// TwinCAT 3 PLC project DMMS_PLC
// ProgramVersion: 3.1.4026.19
// libraries:
//   Tc2_Standard, * (Beckhoff Automation GmbH)
//   Tc2_System, * (Beckhoff Automation GmbH)
//   Tc3_Mc3PlanarMotion, * (Beckhoff Automation GmbH)
//   Tc3_Physics, * (Beckhoff Automation GmbH)
//   Tc3_XPlanarStandard, * (Beckhoff Automation GmbH)
//   Tc3_XPlanarUtility, * (Beckhoff Automation GmbH)
// project tree:
//   DUTs/Communiction/GlobalStatus/ ST_ComIn_GlobalStatus.TcDUT (not stored), ST_ComOut_GlobalStatus.TcDUT (not stored), ST_Com_GlobalStatus.TcDUT (not stored)
//   DUTs/Communiction/Movers/ ST_ComIn_ExportMover.TcDUT, ST_ComOut_ExportMover.TcDUT, ST_PartTrackingData.TcDUT, ST_Com_ExportMover.TcDUT
//   DUTs/Communiction/Station/ ST_ComIn_ExportStation.TcDUT, ST_ComOut_ExportStation.TcDUT, ST_EStationName.TcDUT, ST_ManMov_Station.TcDUT, ST_Com_ExportStation.TcDUT
//   GVLs/ Communication.TcGVL, Debug.TcGVL (not stored), GVL.TcGVL
//   Mover/DUTs/ MoverPositionUnion.TcDUT (not stored), ST_ControlData.TcDUT, ST_EMoverLoadType.TcDUT, ST_ManMov_FreeMove.TcDUT (not stored), ST_ManMov_MoveTrack.TcDUT, ST_ManualMovements.TcDUT (not stored), ST_MoverConfiguration.TcDUT (not stored), ST_ProcessResult.TcDUT (not stored), ST_ProcessTask.TcDUT, ST_ProductData.TcDUT, ST_WellplateParametrization.TcDUT
//   Mover/ FB_ApplicationMover.TcPOU, I_MoverApplication.TcIO
//   / PlcTask.TcTTO (not stored)
//   POUs/ FB_MotionSystem.TcPOU, MAIN.TcPOU
//   Stations/Base/ FB_StationBase.TcPOU, I_Station.TcIO
//   Stations/DUTs/ E_ProcessMode.TcDUT (not stored), ST_EStationProcessState.TcDUT, ST_EStationHandshake.TcDUT (not stored), ST_StationPosition.TcDUT, ST_StationReturn.TcDUT (not stored), ST_VisStationData.TcDUT
//   Stations/ FB_PuncherStation.TcPOU, FB_PuncherSeparateStation.TcPOU (not stored), FB_PuncherBufferStation.TcPOU (not stored)
//   Stations/Helper/ FB_HistoryInfo.TcPOU (not stored)
//   Tracks/Base/ FB_BaseTrack.TcPOU (not stored), I_Track.TcIO (not stored)
//   Tracks/ FB_CloseLoopTrack.TcPOU, FB_UserInteractionTrack.TcPOU (not stored), FB_PipettePreBufferTrack.TcPOU (not stored), FB_PipetteTrack.TcPOU, FB_PipettePostBufferTrack.TcPOU (not stored), FB_PipetteBufferConTrack.TcPOU (not stored), FB_PuncherWellplateTrack.TcPOU (not stored), FB_PuncherBufferTrack.TcPOU, FB_StradeFirstSegTrack.TcPOU (not stored), FB_StradeSecondSegTrack.TcPOU (not stored), FB_PuncherSeperateTrack.TcPOU (not stored)
// real-time tasks:
//   TASK Job Task: cycle default, priority 2
//   TASK MC-Task (MET): cycle T#2ms, priority 3, ADS port 351
//   TASK MC-Task (MPT): cycle T#10ms, priority 4, ADS port 352
//   TASK PlcTask: cycle T#10ms, priority 20, ADS port 353
//   TASK XPlanar Task_0: cycle T#250us, priority 1, ADS port 350
//   TASK XPlanar Task_10: cycle T#250us, priority 5, ADS port 354
// I/O:
//   DEVICE Device 2 (EtherCAT), AmsNetId 192.168.2.44.3.1
//     Term 1 (APS4322-7000) [APS4322-7000 Drive]
//       Term 2 (APS4322-5000) [APS4322-5000 Feedback]
//     Term 3 (APS4322-7000) [APS4322-7000 Drive]
//       Term 4 (APS4322-5000) [APS4322-5000 Feedback]
//     Term 5 (APS4322-7000) [APS4322-7000 Drive]
//       Term 6 (APS4322-5000) [APS4322-5000 Feedback]
//     Term 7 (APS4322-7000) [APS4322-7000 Drive]
//       Term 8 (APS4322-5000) [APS4322-5000 Feedback]
//     Term 9 (APS4322-7000) [APS4322-7000 Drive]
//       Term 10 (APS4322-5000) [APS4322-5000 Feedback]
// variable links:
//   Device 2 (EtherCAT) <-> TcCOM Objects/XPlanar/Part1/APS4322_P1_1
//     Term 1 (APS4322-7000)/APS Comm Inputs/CommStatusWord <-> Data Pointer/MoverCommStatusWord
//     Term 1 (APS4322-7000)/APS Comm Inputs/Data {1..4} <-> Data Pointer/MoverCommDataIn[{0..3}]  (4 links)
//     Term 1 (APS4322-7000)/APS Comm Outputs/CommControlWord <-> Data Pointer/MoverCommControlWord
//     Term 1 (APS4322-7000)/APS Comm Outputs/Data 1 <-> Data Pointer/MoverCommDataOut
//     Term 1 (APS4322-7000)/APS Diagdata/DC Link Voltage <-> Data Pointer/DcLinkVoltage
//     Term 1 (APS4322-7000)/APS Diagdata/Power supply current <-> Data Pointer/PowerSupplyCurrent
//     Term 1 (APS4322-7000)/APS Inputs/StatusWord <-> Data Pointer/PowerUnitStatusWord
//     Term 1 (APS4322-7000)/APS Outputs/ControlWord <-> Data Pointer/PowerUnitControlWord
//     Term 1 (APS4322-7000)/APS Outputs/Current D 0X0 <-> Data Pointer/DCurrentSetPoints[0]
//     Term 1 (APS4322-7000)/APS Outputs/Current D 0X1 <-> Data Pointer/DCurrentSetPoints[1]
//     Term 1 (APS4322-7000)/APS Outputs/Current D 0X2 <-> Data Pointer/DCurrentSetPoints[2]
//     Term 1 (APS4322-7000)/APS Outputs/Current D 1X0 <-> Data Pointer/DCurrentSetPoints[6]
//     Term 1 (APS4322-7000)/APS Outputs/Current D 1X1 <-> Data Pointer/DCurrentSetPoints[7]
//     Term 1 (APS4322-7000)/APS Outputs/Current D 1X2 <-> Data Pointer/DCurrentSetPoints[8]
//     Term 1 (APS4322-7000)/APS Outputs/Current D 2X0 <-> Data Pointer/DCurrentSetPoints[12]
//     Term 1 (APS4322-7000)/APS Outputs/Current D 2X1 <-> Data Pointer/DCurrentSetPoints[13]
//     Term 1 (APS4322-7000)/APS Outputs/Current D 2X2 <-> Data Pointer/DCurrentSetPoints[14]
//     Term 1 (APS4322-7000)/APS Outputs/Current D 3X0 <-> Data Pointer/DCurrentSetPoints[18]
//     Term 1 (APS4322-7000)/APS Outputs/Current D 3X1 <-> Data Pointer/DCurrentSetPoints[19]
//     Term 1 (APS4322-7000)/APS Outputs/Current D 3X2 <-> Data Pointer/DCurrentSetPoints[20]
//     Term 1 (APS4322-7000)/APS Outputs/Current D 0Y0 <-> Data Pointer/DCurrentSetPoints[3]
//     Term 1 (APS4322-7000)/APS Outputs/Current D 0Y1 <-> Data Pointer/DCurrentSetPoints[4]
//     Term 1 (APS4322-7000)/APS Outputs/Current D 0Y2 <-> Data Pointer/DCurrentSetPoints[5]
//     Term 1 (APS4322-7000)/APS Outputs/Current D 1Y0 <-> Data Pointer/DCurrentSetPoints[9]
//     Term 1 (APS4322-7000)/APS Outputs/Current D 1Y1 <-> Data Pointer/DCurrentSetPoints[10]
//     Term 1 (APS4322-7000)/APS Outputs/Current D 1Y2 <-> Data Pointer/DCurrentSetPoints[11]
//     Term 1 (APS4322-7000)/APS Outputs/Current D 2Y0 <-> Data Pointer/DCurrentSetPoints[15]
//     Term 1 (APS4322-7000)/APS Outputs/Current D 2Y1 <-> Data Pointer/DCurrentSetPoints[16]
//     Term 1 (APS4322-7000)/APS Outputs/Current D 2Y2 <-> Data Pointer/DCurrentSetPoints[17]
//     Term 1 (APS4322-7000)/APS Outputs/Current D 3Y0 <-> Data Pointer/DCurrentSetPoints[21]
//     Term 1 (APS4322-7000)/APS Outputs/Current D 3Y1 <-> Data Pointer/DCurrentSetPoints[22]
//     Term 1 (APS4322-7000)/APS Outputs/Current D 3Y2 <-> Data Pointer/DCurrentSetPoints[23]
//     Term 1 (APS4322-7000)/APS Outputs/Current Q 0X0 <-> Data Pointer/QCurrentSetPoints[0]
//     Term 1 (APS4322-7000)/APS Outputs/Current Q 0X1 <-> Data Pointer/QCurrentSetPoints[1]
//     Term 1 (APS4322-7000)/APS Outputs/Current Q 0X2 <-> Data Pointer/QCurrentSetPoints[2]
//     Term 1 (APS4322-7000)/APS Outputs/Current Q 1X0 <-> Data Pointer/QCurrentSetPoints[6]
//     Term 1 (APS4322-7000)/APS Outputs/Current Q 1X1 <-> Data Pointer/QCurrentSetPoints[7]
//     Term 1 (APS4322-7000)/APS Outputs/Current Q 1X2 <-> Data Pointer/QCurrentSetPoints[8]
//     Term 1 (APS4322-7000)/APS Outputs/Current Q 2X0 <-> Data Pointer/QCurrentSetPoints[12]
//     Term 1 (APS4322-7000)/APS Outputs/Current Q 2X1 <-> Data Pointer/QCurrentSetPoints[13]
//     Term 1 (APS4322-7000)/APS Outputs/Current Q 2X2 <-> Data Pointer/QCurrentSetPoints[14]
//     Term 1 (APS4322-7000)/APS Outputs/Current Q 3X0 <-> Data Pointer/QCurrentSetPoints[18]
//     Term 1 (APS4322-7000)/APS Outputs/Current Q 3X1 <-> Data Pointer/QCurrentSetPoints[19]
//     Term 1 (APS4322-7000)/APS Outputs/Current Q 3X2 <-> Data Pointer/QCurrentSetPoints[20]
//     Term 1 (APS4322-7000)/APS Outputs/Current Q 0Y0 <-> Data Pointer/QCurrentSetPoints[3]
//     Term 1 (APS4322-7000)/APS Outputs/Current Q 0Y1 <-> Data Pointer/QCurrentSetPoints[4]
//     Term 1 (APS4322-7000)/APS Outputs/Current Q 0Y2 <-> Data Pointer/QCurrentSetPoints[5]
//     Term 1 (APS4322-7000)/APS Outputs/Current Q 1Y0 <-> Data Pointer/QCurrentSetPoints[9]
//     Term 1 (APS4322-7000)/APS Outputs/Current Q 1Y1 <-> Data Pointer/QCurrentSetPoints[10]
//     Term 1 (APS4322-7000)/APS Outputs/Current Q 1Y2 <-> Data Pointer/QCurrentSetPoints[11]
//     Term 1 (APS4322-7000)/APS Outputs/Current Q 2Y0 <-> Data Pointer/QCurrentSetPoints[15]
//     Term 1 (APS4322-7000)/APS Outputs/Current Q 2Y1 <-> Data Pointer/QCurrentSetPoints[16]
//     Term 1 (APS4322-7000)/APS Outputs/Current Q 2Y2 <-> Data Pointer/QCurrentSetPoints[17]
//     Term 1 (APS4322-7000)/APS Outputs/Current Q 3Y0 <-> Data Pointer/QCurrentSetPoints[21]
//     Term 1 (APS4322-7000)/APS Outputs/Current Q 3Y1 <-> Data Pointer/QCurrentSetPoints[22]
//     Term 1 (APS4322-7000)/APS Outputs/Current Q 3Y2 <-> Data Pointer/QCurrentSetPoints[23]
//     Term 1 (APS4322-7000)/APS Outputs/PhiE 0X0 <-> Data Pointer/PhiSetPoints[0]
//     Term 1 (APS4322-7000)/APS Outputs/PhiE 0X1 <-> Data Pointer/PhiSetPoints[1]
//     Term 1 (APS4322-7000)/APS Outputs/PhiE 0X2 <-> Data Pointer/PhiSetPoints[2]
//     Term 1 (APS4322-7000)/APS Outputs/PhiE 1X0 <-> Data Pointer/PhiSetPoints[6]
//     Term 1 (APS4322-7000)/APS Outputs/PhiE 1X1 <-> Data Pointer/PhiSetPoints[7]
//     Term 1 (APS4322-7000)/APS Outputs/PhiE 1X2 <-> Data Pointer/PhiSetPoints[8]
//     Term 1 (APS4322-7000)/APS Outputs/PhiE 2X0 <-> Data Pointer/PhiSetPoints[12]
//     Term 1 (APS4322-7000)/APS Outputs/PhiE 2X1 <-> Data Pointer/PhiSetPoints[13]
//     Term 1 (APS4322-7000)/APS Outputs/PhiE 2X2 <-> Data Pointer/PhiSetPoints[14]
//     Term 1 (APS4322-7000)/APS Outputs/PhiE 3X0 <-> Data Pointer/PhiSetPoints[18]
//     Term 1 (APS4322-7000)/APS Outputs/PhiE 3X1 <-> Data Pointer/PhiSetPoints[19]
//     Term 1 (APS4322-7000)/APS Outputs/PhiE 3X2 <-> Data Pointer/PhiSetPoints[20]
//     Term 1 (APS4322-7000)/APS Outputs/PhiE 0Y0 <-> Data Pointer/PhiSetPoints[3]
//     Term 1 (APS4322-7000)/APS Outputs/PhiE 0Y1 <-> Data Pointer/PhiSetPoints[4]
//     Term 1 (APS4322-7000)/APS Outputs/PhiE 0Y2 <-> Data Pointer/PhiSetPoints[5]
//     Term 1 (APS4322-7000)/APS Outputs/PhiE 1Y0 <-> Data Pointer/PhiSetPoints[9]
//     Term 1 (APS4322-7000)/APS Outputs/PhiE 1Y1 <-> Data Pointer/PhiSetPoints[10]
//     Term 1 (APS4322-7000)/APS Outputs/PhiE 1Y2 <-> Data Pointer/PhiSetPoints[11]
//     Term 1 (APS4322-7000)/APS Outputs/PhiE 2Y0 <-> Data Pointer/PhiSetPoints[15]
//     Term 1 (APS4322-7000)/APS Outputs/PhiE 2Y1 <-> Data Pointer/PhiSetPoints[16]
//     Term 1 (APS4322-7000)/APS Outputs/PhiE 2Y2 <-> Data Pointer/PhiSetPoints[17]
//     Term 1 (APS4322-7000)/APS Outputs/PhiE 3Y0 <-> Data Pointer/PhiSetPoints[21]
//     Term 1 (APS4322-7000)/APS Outputs/PhiE 3Y1 <-> Data Pointer/PhiSetPoints[22]
//     Term 1 (APS4322-7000)/APS Outputs/PhiE 3Y2 <-> Data Pointer/PhiSetPoints[23]
//     Term 1 (APS4322-7000)/Term 2 (APS4322-5000)/FB Inputs/A{0..8 step 2} X-Field <-> Data Pointer/HallSensorFieldsXYZ[{0..12 step 3}]  (5 links)
//     Term 1 (APS4322-7000)/Term 2 (APS4322-5000)/FB Inputs/A{0..8 step 2} Y-Field <-> Data Pointer/HallSensorFieldsXYZ[{1..13 step 3}]  (5 links)
//     Term 1 (APS4322-7000)/Term 2 (APS4322-5000)/FB Inputs/A{0..8 step 2} Z-Field <-> Data Pointer/HallSensorFieldsXYZ[{2..14 step 3}]  (5 links)
//     Term 1 (APS4322-7000)/Term 2 (APS4322-5000)/FB Inputs/B{1..9 step 2} X-Field <-> Data Pointer/HallSensorFieldsXYZ[{15..27 step 3}]  (5 links)
//     Term 1 (APS4322-7000)/Term 2 (APS4322-5000)/FB Inputs/B{1..9 step 2} Y-Field <-> Data Pointer/HallSensorFieldsXYZ[{16..28 step 3}]  (5 links)
//     Term 1 (APS4322-7000)/Term 2 (APS4322-5000)/FB Inputs/B{1..9 step 2} Z-Field <-> Data Pointer/HallSensorFieldsXYZ[{17..29 step 3}]  (5 links)
//     Term 1 (APS4322-7000)/Term 2 (APS4322-5000)/FB Inputs/C{0..8 step 2} X-Field <-> Data Pointer/HallSensorFieldsXYZ[{30..42 step 3}]  (5 links)
//     Term 1 (APS4322-7000)/Term 2 (APS4322-5000)/FB Inputs/C{0..8 step 2} Y-Field <-> Data Pointer/HallSensorFieldsXYZ[{31..43 step 3}]  (5 links)
//     Term 1 (APS4322-7000)/Term 2 (APS4322-5000)/FB Inputs/C{0..8 step 2} Z-Field <-> Data Pointer/HallSensorFieldsXYZ[{32..44 step 3}]  (5 links)
//     Term 1 (APS4322-7000)/Term 2 (APS4322-5000)/FB Inputs/D{1..9 step 2} X-Field <-> Data Pointer/HallSensorFieldsXYZ[{45..57 step 3}]  (5 links)
//     Term 1 (APS4322-7000)/Term 2 (APS4322-5000)/FB Inputs/D{1..9 step 2} Y-Field <-> Data Pointer/HallSensorFieldsXYZ[{46..58 step 3}]  (5 links)
//     Term 1 (APS4322-7000)/Term 2 (APS4322-5000)/FB Inputs/D{1..9 step 2} Z-Field <-> Data Pointer/HallSensorFieldsXYZ[{47..59 step 3}]  (5 links)
//     Term 1 (APS4322-7000)/Term 2 (APS4322-5000)/FB Inputs/E{0..8 step 2} X-Field <-> Data Pointer/HallSensorFieldsXYZ[{60..72 step 3}]  (5 links)
//     Term 1 (APS4322-7000)/Term 2 (APS4322-5000)/FB Inputs/E{0..8 step 2} Y-Field <-> Data Pointer/HallSensorFieldsXYZ[{61..73 step 3}]  (5 links)
//     Term 1 (APS4322-7000)/Term 2 (APS4322-5000)/FB Inputs/E{0..8 step 2} Z-Field <-> Data Pointer/HallSensorFieldsXYZ[{62..74 step 3}]  (5 links)
//     Term 1 (APS4322-7000)/Term 2 (APS4322-5000)/FB Inputs/F{1..9 step 2} X-Field <-> Data Pointer/HallSensorFieldsXYZ[{75..87 step 3}]  (5 links)
//     Term 1 (APS4322-7000)/Term 2 (APS4322-5000)/FB Inputs/F{1..9 step 2} Y-Field <-> Data Pointer/HallSensorFieldsXYZ[{76..88 step 3}]  (5 links)
//     Term 1 (APS4322-7000)/Term 2 (APS4322-5000)/FB Inputs/F{1..9 step 2} Z-Field <-> Data Pointer/HallSensorFieldsXYZ[{77..89 step 3}]  (5 links)
//     Term 1 (APS4322-7000)/Term 2 (APS4322-5000)/FB Inputs/G{0..8 step 2} X-Field <-> Data Pointer/HallSensorFieldsXYZ[{90..102 step 3}]  (5 links)
//     Term 1 (APS4322-7000)/Term 2 (APS4322-5000)/FB Inputs/G{0..8 step 2} Y-Field <-> Data Pointer/HallSensorFieldsXYZ[{91..103 step 3}]  (5 links)
//     Term 1 (APS4322-7000)/Term 2 (APS4322-5000)/FB Inputs/G{0..8 step 2} Z-Field <-> Data Pointer/HallSensorFieldsXYZ[{92..104 step 3}]  (5 links)
//     Term 1 (APS4322-7000)/Term 2 (APS4322-5000)/FB Inputs/H{1..9 step 2} X-Field <-> Data Pointer/HallSensorFieldsXYZ[{105..117 step 3}]  (5 links)
//     Term 1 (APS4322-7000)/Term 2 (APS4322-5000)/FB Inputs/H{1..9 step 2} Y-Field <-> Data Pointer/HallSensorFieldsXYZ[{106..118 step 3}]  (5 links)
//     Term 1 (APS4322-7000)/Term 2 (APS4322-5000)/FB Inputs/H{1..9 step 2} Z-Field <-> Data Pointer/HallSensorFieldsXYZ[{107..119 step 3}]  (5 links)
//     Term 1 (APS4322-7000)/Term 2 (APS4322-5000)/FB Inputs/I{0..8 step 2} X-Field <-> Data Pointer/HallSensorFieldsXYZ[{120..132 step 3}]  (5 links)
//     Term 1 (APS4322-7000)/Term 2 (APS4322-5000)/FB Inputs/I{0..8 step 2} Y-Field <-> Data Pointer/HallSensorFieldsXYZ[{121..133 step 3}]  (5 links)
//     Term 1 (APS4322-7000)/Term 2 (APS4322-5000)/FB Inputs/I{0..8 step 2} Z-Field <-> Data Pointer/HallSensorFieldsXYZ[{122..134 step 3}]  (5 links)
//     Term 1 (APS4322-7000)/Term 2 (APS4322-5000)/FB Inputs/J{1..9 step 2} X-Field <-> Data Pointer/HallSensorFieldsXYZ[{135..147 step 3}]  (5 links)
//     Term 1 (APS4322-7000)/Term 2 (APS4322-5000)/FB Inputs/J{1..9 step 2} Y-Field <-> Data Pointer/HallSensorFieldsXYZ[{136..148 step 3}]  (5 links)
//     Term 1 (APS4322-7000)/Term 2 (APS4322-5000)/FB Inputs/J{1..9 step 2} Z-Field <-> Data Pointer/HallSensorFieldsXYZ[{137..149 step 3}]  (5 links)
//     Term 1 (APS4322-7000)/Term 2 (APS4322-5000)/FB Inputs/Status <-> Data Pointer/FeedbackStatus
//   Device 2 (EtherCAT) <-> TcCOM Objects/XPlanar/Part1/APS4322_P1_2
//     Term 3 (APS4322-7000)/APS Comm Inputs/CommStatusWord <-> Data Pointer/MoverCommStatusWord
//     Term 3 (APS4322-7000)/APS Comm Inputs/Data {1..4} <-> Data Pointer/MoverCommDataIn[{0..3}]  (4 links)
//     Term 3 (APS4322-7000)/APS Comm Outputs/CommControlWord <-> Data Pointer/MoverCommControlWord
//     Term 3 (APS4322-7000)/APS Comm Outputs/Data 1 <-> Data Pointer/MoverCommDataOut
//     Term 3 (APS4322-7000)/APS Diagdata/DC Link Voltage <-> Data Pointer/DcLinkVoltage
//     Term 3 (APS4322-7000)/APS Diagdata/Power supply current <-> Data Pointer/PowerSupplyCurrent
//     Term 3 (APS4322-7000)/APS Inputs/StatusWord <-> Data Pointer/PowerUnitStatusWord
//     Term 3 (APS4322-7000)/APS Outputs/ControlWord <-> Data Pointer/PowerUnitControlWord
//     Term 3 (APS4322-7000)/APS Outputs/Current D 0X0 <-> Data Pointer/DCurrentSetPoints[0]
//     Term 3 (APS4322-7000)/APS Outputs/Current D 0X1 <-> Data Pointer/DCurrentSetPoints[1]
//     Term 3 (APS4322-7000)/APS Outputs/Current D 0X2 <-> Data Pointer/DCurrentSetPoints[2]
//     Term 3 (APS4322-7000)/APS Outputs/Current D 1X0 <-> Data Pointer/DCurrentSetPoints[6]
//     Term 3 (APS4322-7000)/APS Outputs/Current D 1X1 <-> Data Pointer/DCurrentSetPoints[7]
//     Term 3 (APS4322-7000)/APS Outputs/Current D 1X2 <-> Data Pointer/DCurrentSetPoints[8]
//     Term 3 (APS4322-7000)/APS Outputs/Current D 2X0 <-> Data Pointer/DCurrentSetPoints[12]
//     Term 3 (APS4322-7000)/APS Outputs/Current D 2X1 <-> Data Pointer/DCurrentSetPoints[13]
//     Term 3 (APS4322-7000)/APS Outputs/Current D 2X2 <-> Data Pointer/DCurrentSetPoints[14]
//     Term 3 (APS4322-7000)/APS Outputs/Current D 3X0 <-> Data Pointer/DCurrentSetPoints[18]
//     Term 3 (APS4322-7000)/APS Outputs/Current D 3X1 <-> Data Pointer/DCurrentSetPoints[19]
//     Term 3 (APS4322-7000)/APS Outputs/Current D 3X2 <-> Data Pointer/DCurrentSetPoints[20]
//     Term 3 (APS4322-7000)/APS Outputs/Current D 0Y0 <-> Data Pointer/DCurrentSetPoints[3]
//     Term 3 (APS4322-7000)/APS Outputs/Current D 0Y1 <-> Data Pointer/DCurrentSetPoints[4]
//     Term 3 (APS4322-7000)/APS Outputs/Current D 0Y2 <-> Data Pointer/DCurrentSetPoints[5]
//     Term 3 (APS4322-7000)/APS Outputs/Current D 1Y0 <-> Data Pointer/DCurrentSetPoints[9]
//     Term 3 (APS4322-7000)/APS Outputs/Current D 1Y1 <-> Data Pointer/DCurrentSetPoints[10]
//     Term 3 (APS4322-7000)/APS Outputs/Current D 1Y2 <-> Data Pointer/DCurrentSetPoints[11]
//     Term 3 (APS4322-7000)/APS Outputs/Current D 2Y0 <-> Data Pointer/DCurrentSetPoints[15]
//     Term 3 (APS4322-7000)/APS Outputs/Current D 2Y1 <-> Data Pointer/DCurrentSetPoints[16]
//     Term 3 (APS4322-7000)/APS Outputs/Current D 2Y2 <-> Data Pointer/DCurrentSetPoints[17]
//     Term 3 (APS4322-7000)/APS Outputs/Current D 3Y0 <-> Data Pointer/DCurrentSetPoints[21]
//     Term 3 (APS4322-7000)/APS Outputs/Current D 3Y1 <-> Data Pointer/DCurrentSetPoints[22]
//     Term 3 (APS4322-7000)/APS Outputs/Current D 3Y2 <-> Data Pointer/DCurrentSetPoints[23]
//     Term 3 (APS4322-7000)/APS Outputs/Current Q 0X0 <-> Data Pointer/QCurrentSetPoints[0]
//     Term 3 (APS4322-7000)/APS Outputs/Current Q 0X1 <-> Data Pointer/QCurrentSetPoints[1]
//     Term 3 (APS4322-7000)/APS Outputs/Current Q 0X2 <-> Data Pointer/QCurrentSetPoints[2]
//     Term 3 (APS4322-7000)/APS Outputs/Current Q 1X0 <-> Data Pointer/QCurrentSetPoints[6]
//     Term 3 (APS4322-7000)/APS Outputs/Current Q 1X1 <-> Data Pointer/QCurrentSetPoints[7]
//     Term 3 (APS4322-7000)/APS Outputs/Current Q 1X2 <-> Data Pointer/QCurrentSetPoints[8]
//     Term 3 (APS4322-7000)/APS Outputs/Current Q 2X0 <-> Data Pointer/QCurrentSetPoints[12]
//     Term 3 (APS4322-7000)/APS Outputs/Current Q 2X1 <-> Data Pointer/QCurrentSetPoints[13]
//     Term 3 (APS4322-7000)/APS Outputs/Current Q 2X2 <-> Data Pointer/QCurrentSetPoints[14]
//     Term 3 (APS4322-7000)/APS Outputs/Current Q 3X0 <-> Data Pointer/QCurrentSetPoints[18]
//     Term 3 (APS4322-7000)/APS Outputs/Current Q 3X1 <-> Data Pointer/QCurrentSetPoints[19]
//     Term 3 (APS4322-7000)/APS Outputs/Current Q 3X2 <-> Data Pointer/QCurrentSetPoints[20]
//     Term 3 (APS4322-7000)/APS Outputs/Current Q 0Y0 <-> Data Pointer/QCurrentSetPoints[3]
//     Term 3 (APS4322-7000)/APS Outputs/Current Q 0Y1 <-> Data Pointer/QCurrentSetPoints[4]
//     Term 3 (APS4322-7000)/APS Outputs/Current Q 0Y2 <-> Data Pointer/QCurrentSetPoints[5]
//     Term 3 (APS4322-7000)/APS Outputs/Current Q 1Y0 <-> Data Pointer/QCurrentSetPoints[9]
//     Term 3 (APS4322-7000)/APS Outputs/Current Q 1Y1 <-> Data Pointer/QCurrentSetPoints[10]
//     Term 3 (APS4322-7000)/APS Outputs/Current Q 1Y2 <-> Data Pointer/QCurrentSetPoints[11]
//     Term 3 (APS4322-7000)/APS Outputs/Current Q 2Y0 <-> Data Pointer/QCurrentSetPoints[15]
//     Term 3 (APS4322-7000)/APS Outputs/Current Q 2Y1 <-> Data Pointer/QCurrentSetPoints[16]
//     Term 3 (APS4322-7000)/APS Outputs/Current Q 2Y2 <-> Data Pointer/QCurrentSetPoints[17]
//     Term 3 (APS4322-7000)/APS Outputs/Current Q 3Y0 <-> Data Pointer/QCurrentSetPoints[21]
//     Term 3 (APS4322-7000)/APS Outputs/Current Q 3Y1 <-> Data Pointer/QCurrentSetPoints[22]
//     Term 3 (APS4322-7000)/APS Outputs/Current Q 3Y2 <-> Data Pointer/QCurrentSetPoints[23]
//     Term 3 (APS4322-7000)/APS Outputs/PhiE 0X0 <-> Data Pointer/PhiSetPoints[0]
//     Term 3 (APS4322-7000)/APS Outputs/PhiE 0X1 <-> Data Pointer/PhiSetPoints[1]
//     Term 3 (APS4322-7000)/APS Outputs/PhiE 0X2 <-> Data Pointer/PhiSetPoints[2]
//     Term 3 (APS4322-7000)/APS Outputs/PhiE 1X0 <-> Data Pointer/PhiSetPoints[6]
//     Term 3 (APS4322-7000)/APS Outputs/PhiE 1X1 <-> Data Pointer/PhiSetPoints[7]
//     Term 3 (APS4322-7000)/APS Outputs/PhiE 1X2 <-> Data Pointer/PhiSetPoints[8]
//     Term 3 (APS4322-7000)/APS Outputs/PhiE 2X0 <-> Data Pointer/PhiSetPoints[12]
//     Term 3 (APS4322-7000)/APS Outputs/PhiE 2X1 <-> Data Pointer/PhiSetPoints[13]
//     Term 3 (APS4322-7000)/APS Outputs/PhiE 2X2 <-> Data Pointer/PhiSetPoints[14]
//     Term 3 (APS4322-7000)/APS Outputs/PhiE 3X0 <-> Data Pointer/PhiSetPoints[18]
//     Term 3 (APS4322-7000)/APS Outputs/PhiE 3X1 <-> Data Pointer/PhiSetPoints[19]
//     Term 3 (APS4322-7000)/APS Outputs/PhiE 3X2 <-> Data Pointer/PhiSetPoints[20]
//     Term 3 (APS4322-7000)/APS Outputs/PhiE 0Y0 <-> Data Pointer/PhiSetPoints[3]
//     Term 3 (APS4322-7000)/APS Outputs/PhiE 0Y1 <-> Data Pointer/PhiSetPoints[4]
//     Term 3 (APS4322-7000)/APS Outputs/PhiE 0Y2 <-> Data Pointer/PhiSetPoints[5]
//     Term 3 (APS4322-7000)/APS Outputs/PhiE 1Y0 <-> Data Pointer/PhiSetPoints[9]
//     Term 3 (APS4322-7000)/APS Outputs/PhiE 1Y1 <-> Data Pointer/PhiSetPoints[10]
//     Term 3 (APS4322-7000)/APS Outputs/PhiE 1Y2 <-> Data Pointer/PhiSetPoints[11]
//     Term 3 (APS4322-7000)/APS Outputs/PhiE 2Y0 <-> Data Pointer/PhiSetPoints[15]
//     Term 3 (APS4322-7000)/APS Outputs/PhiE 2Y1 <-> Data Pointer/PhiSetPoints[16]
//     Term 3 (APS4322-7000)/APS Outputs/PhiE 2Y2 <-> Data Pointer/PhiSetPoints[17]
//     Term 3 (APS4322-7000)/APS Outputs/PhiE 3Y0 <-> Data Pointer/PhiSetPoints[21]
//     Term 3 (APS4322-7000)/APS Outputs/PhiE 3Y1 <-> Data Pointer/PhiSetPoints[22]
//     Term 3 (APS4322-7000)/APS Outputs/PhiE 3Y2 <-> Data Pointer/PhiSetPoints[23]
//     Term 3 (APS4322-7000)/Term 4 (APS4322-5000)/FB Inputs/A{0..8 step 2} X-Field <-> Data Pointer/HallSensorFieldsXYZ[{0..12 step 3}]  (5 links)
//     Term 3 (APS4322-7000)/Term 4 (APS4322-5000)/FB Inputs/A{0..8 step 2} Y-Field <-> Data Pointer/HallSensorFieldsXYZ[{1..13 step 3}]  (5 links)
//     Term 3 (APS4322-7000)/Term 4 (APS4322-5000)/FB Inputs/A{0..8 step 2} Z-Field <-> Data Pointer/HallSensorFieldsXYZ[{2..14 step 3}]  (5 links)
//     Term 3 (APS4322-7000)/Term 4 (APS4322-5000)/FB Inputs/B{1..9 step 2} X-Field <-> Data Pointer/HallSensorFieldsXYZ[{15..27 step 3}]  (5 links)
//     Term 3 (APS4322-7000)/Term 4 (APS4322-5000)/FB Inputs/B{1..9 step 2} Y-Field <-> Data Pointer/HallSensorFieldsXYZ[{16..28 step 3}]  (5 links)
//     Term 3 (APS4322-7000)/Term 4 (APS4322-5000)/FB Inputs/B{1..9 step 2} Z-Field <-> Data Pointer/HallSensorFieldsXYZ[{17..29 step 3}]  (5 links)
//     Term 3 (APS4322-7000)/Term 4 (APS4322-5000)/FB Inputs/C{0..8 step 2} X-Field <-> Data Pointer/HallSensorFieldsXYZ[{30..42 step 3}]  (5 links)
//     Term 3 (APS4322-7000)/Term 4 (APS4322-5000)/FB Inputs/C{0..8 step 2} Y-Field <-> Data Pointer/HallSensorFieldsXYZ[{31..43 step 3}]  (5 links)
//     Term 3 (APS4322-7000)/Term 4 (APS4322-5000)/FB Inputs/C{0..8 step 2} Z-Field <-> Data Pointer/HallSensorFieldsXYZ[{32..44 step 3}]  (5 links)
//     Term 3 (APS4322-7000)/Term 4 (APS4322-5000)/FB Inputs/D{1..9 step 2} X-Field <-> Data Pointer/HallSensorFieldsXYZ[{45..57 step 3}]  (5 links)
//     Term 3 (APS4322-7000)/Term 4 (APS4322-5000)/FB Inputs/D{1..9 step 2} Y-Field <-> Data Pointer/HallSensorFieldsXYZ[{46..58 step 3}]  (5 links)
//     Term 3 (APS4322-7000)/Term 4 (APS4322-5000)/FB Inputs/D{1..9 step 2} Z-Field <-> Data Pointer/HallSensorFieldsXYZ[{47..59 step 3}]  (5 links)
//     Term 3 (APS4322-7000)/Term 4 (APS4322-5000)/FB Inputs/E{0..8 step 2} X-Field <-> Data Pointer/HallSensorFieldsXYZ[{60..72 step 3}]  (5 links)
//     Term 3 (APS4322-7000)/Term 4 (APS4322-5000)/FB Inputs/E{0..8 step 2} Y-Field <-> Data Pointer/HallSensorFieldsXYZ[{61..73 step 3}]  (5 links)
//     Term 3 (APS4322-7000)/Term 4 (APS4322-5000)/FB Inputs/E{0..8 step 2} Z-Field <-> Data Pointer/HallSensorFieldsXYZ[{62..74 step 3}]  (5 links)
//     Term 3 (APS4322-7000)/Term 4 (APS4322-5000)/FB Inputs/F{1..9 step 2} X-Field <-> Data Pointer/HallSensorFieldsXYZ[{75..87 step 3}]  (5 links)
//     Term 3 (APS4322-7000)/Term 4 (APS4322-5000)/FB Inputs/F{1..9 step 2} Y-Field <-> Data Pointer/HallSensorFieldsXYZ[{76..88 step 3}]  (5 links)
//     Term 3 (APS4322-7000)/Term 4 (APS4322-5000)/FB Inputs/F{1..9 step 2} Z-Field <-> Data Pointer/HallSensorFieldsXYZ[{77..89 step 3}]  (5 links)
//     Term 3 (APS4322-7000)/Term 4 (APS4322-5000)/FB Inputs/G{0..8 step 2} X-Field <-> Data Pointer/HallSensorFieldsXYZ[{90..102 step 3}]  (5 links)
//     Term 3 (APS4322-7000)/Term 4 (APS4322-5000)/FB Inputs/G{0..8 step 2} Y-Field <-> Data Pointer/HallSensorFieldsXYZ[{91..103 step 3}]  (5 links)
//     Term 3 (APS4322-7000)/Term 4 (APS4322-5000)/FB Inputs/G{0..8 step 2} Z-Field <-> Data Pointer/HallSensorFieldsXYZ[{92..104 step 3}]  (5 links)
//     Term 3 (APS4322-7000)/Term 4 (APS4322-5000)/FB Inputs/H{1..9 step 2} X-Field <-> Data Pointer/HallSensorFieldsXYZ[{105..117 step 3}]  (5 links)
//     Term 3 (APS4322-7000)/Term 4 (APS4322-5000)/FB Inputs/H{1..9 step 2} Y-Field <-> Data Pointer/HallSensorFieldsXYZ[{106..118 step 3}]  (5 links)
//     Term 3 (APS4322-7000)/Term 4 (APS4322-5000)/FB Inputs/H{1..9 step 2} Z-Field <-> Data Pointer/HallSensorFieldsXYZ[{107..119 step 3}]  (5 links)
//     Term 3 (APS4322-7000)/Term 4 (APS4322-5000)/FB Inputs/I{0..8 step 2} X-Field <-> Data Pointer/HallSensorFieldsXYZ[{120..132 step 3}]  (5 links)
//     Term 3 (APS4322-7000)/Term 4 (APS4322-5000)/FB Inputs/I{0..8 step 2} Y-Field <-> Data Pointer/HallSensorFieldsXYZ[{121..133 step 3}]  (5 links)
//     Term 3 (APS4322-7000)/Term 4 (APS4322-5000)/FB Inputs/I{0..8 step 2} Z-Field <-> Data Pointer/HallSensorFieldsXYZ[{122..134 step 3}]  (5 links)
//     Term 3 (APS4322-7000)/Term 4 (APS4322-5000)/FB Inputs/J{1..9 step 2} X-Field <-> Data Pointer/HallSensorFieldsXYZ[{135..147 step 3}]  (5 links)
//     Term 3 (APS4322-7000)/Term 4 (APS4322-5000)/FB Inputs/J{1..9 step 2} Y-Field <-> Data Pointer/HallSensorFieldsXYZ[{136..148 step 3}]  (5 links)
//     Term 3 (APS4322-7000)/Term 4 (APS4322-5000)/FB Inputs/J{1..9 step 2} Z-Field <-> Data Pointer/HallSensorFieldsXYZ[{137..149 step 3}]  (5 links)
//     Term 3 (APS4322-7000)/Term 4 (APS4322-5000)/FB Inputs/Status <-> Data Pointer/FeedbackStatus
//   Device 2 (EtherCAT) <-> TcCOM Objects/XPlanar/Part1/APS4322_P1_3
//     Term 5 (APS4322-7000)/APS Comm Inputs/CommStatusWord <-> Data Pointer/MoverCommStatusWord
//     Term 5 (APS4322-7000)/APS Comm Inputs/Data {1..4} <-> Data Pointer/MoverCommDataIn[{0..3}]  (4 links)
//     Term 5 (APS4322-7000)/APS Comm Outputs/CommControlWord <-> Data Pointer/MoverCommControlWord
//     Term 5 (APS4322-7000)/APS Comm Outputs/Data 1 <-> Data Pointer/MoverCommDataOut
//     Term 5 (APS4322-7000)/APS Diagdata/DC Link Voltage <-> Data Pointer/DcLinkVoltage
//     Term 5 (APS4322-7000)/APS Diagdata/Power supply current <-> Data Pointer/PowerSupplyCurrent
//     Term 5 (APS4322-7000)/APS Inputs/StatusWord <-> Data Pointer/PowerUnitStatusWord
//     Term 5 (APS4322-7000)/APS Outputs/ControlWord <-> Data Pointer/PowerUnitControlWord
//     Term 5 (APS4322-7000)/APS Outputs/Current D 0X0 <-> Data Pointer/DCurrentSetPoints[0]
//     Term 5 (APS4322-7000)/APS Outputs/Current D 0X1 <-> Data Pointer/DCurrentSetPoints[1]
//     Term 5 (APS4322-7000)/APS Outputs/Current D 0X2 <-> Data Pointer/DCurrentSetPoints[2]
//     Term 5 (APS4322-7000)/APS Outputs/Current D 1X0 <-> Data Pointer/DCurrentSetPoints[6]
//     Term 5 (APS4322-7000)/APS Outputs/Current D 1X1 <-> Data Pointer/DCurrentSetPoints[7]
//     Term 5 (APS4322-7000)/APS Outputs/Current D 1X2 <-> Data Pointer/DCurrentSetPoints[8]
//     Term 5 (APS4322-7000)/APS Outputs/Current D 2X0 <-> Data Pointer/DCurrentSetPoints[12]
//     Term 5 (APS4322-7000)/APS Outputs/Current D 2X1 <-> Data Pointer/DCurrentSetPoints[13]
//     Term 5 (APS4322-7000)/APS Outputs/Current D 2X2 <-> Data Pointer/DCurrentSetPoints[14]
//     Term 5 (APS4322-7000)/APS Outputs/Current D 3X0 <-> Data Pointer/DCurrentSetPoints[18]
//     Term 5 (APS4322-7000)/APS Outputs/Current D 3X1 <-> Data Pointer/DCurrentSetPoints[19]
//     Term 5 (APS4322-7000)/APS Outputs/Current D 3X2 <-> Data Pointer/DCurrentSetPoints[20]
//     Term 5 (APS4322-7000)/APS Outputs/Current D 0Y0 <-> Data Pointer/DCurrentSetPoints[3]
//     Term 5 (APS4322-7000)/APS Outputs/Current D 0Y1 <-> Data Pointer/DCurrentSetPoints[4]
//     Term 5 (APS4322-7000)/APS Outputs/Current D 0Y2 <-> Data Pointer/DCurrentSetPoints[5]
//     Term 5 (APS4322-7000)/APS Outputs/Current D 1Y0 <-> Data Pointer/DCurrentSetPoints[9]
//     Term 5 (APS4322-7000)/APS Outputs/Current D 1Y1 <-> Data Pointer/DCurrentSetPoints[10]
//     Term 5 (APS4322-7000)/APS Outputs/Current D 1Y2 <-> Data Pointer/DCurrentSetPoints[11]
//     Term 5 (APS4322-7000)/APS Outputs/Current D 2Y0 <-> Data Pointer/DCurrentSetPoints[15]
//     Term 5 (APS4322-7000)/APS Outputs/Current D 2Y1 <-> Data Pointer/DCurrentSetPoints[16]
//     Term 5 (APS4322-7000)/APS Outputs/Current D 2Y2 <-> Data Pointer/DCurrentSetPoints[17]
//     Term 5 (APS4322-7000)/APS Outputs/Current D 3Y0 <-> Data Pointer/DCurrentSetPoints[21]
//     Term 5 (APS4322-7000)/APS Outputs/Current D 3Y1 <-> Data Pointer/DCurrentSetPoints[22]
//     Term 5 (APS4322-7000)/APS Outputs/Current D 3Y2 <-> Data Pointer/DCurrentSetPoints[23]
//     Term 5 (APS4322-7000)/APS Outputs/Current Q 0X0 <-> Data Pointer/QCurrentSetPoints[0]
//     Term 5 (APS4322-7000)/APS Outputs/Current Q 0X1 <-> Data Pointer/QCurrentSetPoints[1]
//     Term 5 (APS4322-7000)/APS Outputs/Current Q 0X2 <-> Data Pointer/QCurrentSetPoints[2]
//     Term 5 (APS4322-7000)/APS Outputs/Current Q 1X0 <-> Data Pointer/QCurrentSetPoints[6]
//     Term 5 (APS4322-7000)/APS Outputs/Current Q 1X1 <-> Data Pointer/QCurrentSetPoints[7]
//     Term 5 (APS4322-7000)/APS Outputs/Current Q 1X2 <-> Data Pointer/QCurrentSetPoints[8]
//     Term 5 (APS4322-7000)/APS Outputs/Current Q 2X0 <-> Data Pointer/QCurrentSetPoints[12]
//     Term 5 (APS4322-7000)/APS Outputs/Current Q 2X1 <-> Data Pointer/QCurrentSetPoints[13]
//     Term 5 (APS4322-7000)/APS Outputs/Current Q 2X2 <-> Data Pointer/QCurrentSetPoints[14]
//     Term 5 (APS4322-7000)/APS Outputs/Current Q 3X0 <-> Data Pointer/QCurrentSetPoints[18]
//     Term 5 (APS4322-7000)/APS Outputs/Current Q 3X1 <-> Data Pointer/QCurrentSetPoints[19]
//     Term 5 (APS4322-7000)/APS Outputs/Current Q 3X2 <-> Data Pointer/QCurrentSetPoints[20]
//     Term 5 (APS4322-7000)/APS Outputs/Current Q 0Y0 <-> Data Pointer/QCurrentSetPoints[3]
//     Term 5 (APS4322-7000)/APS Outputs/Current Q 0Y1 <-> Data Pointer/QCurrentSetPoints[4]
//     Term 5 (APS4322-7000)/APS Outputs/Current Q 0Y2 <-> Data Pointer/QCurrentSetPoints[5]
//     Term 5 (APS4322-7000)/APS Outputs/Current Q 1Y0 <-> Data Pointer/QCurrentSetPoints[9]
//     Term 5 (APS4322-7000)/APS Outputs/Current Q 1Y1 <-> Data Pointer/QCurrentSetPoints[10]
//     Term 5 (APS4322-7000)/APS Outputs/Current Q 1Y2 <-> Data Pointer/QCurrentSetPoints[11]
//     Term 5 (APS4322-7000)/APS Outputs/Current Q 2Y0 <-> Data Pointer/QCurrentSetPoints[15]
//     Term 5 (APS4322-7000)/APS Outputs/Current Q 2Y1 <-> Data Pointer/QCurrentSetPoints[16]
//     Term 5 (APS4322-7000)/APS Outputs/Current Q 2Y2 <-> Data Pointer/QCurrentSetPoints[17]
//     Term 5 (APS4322-7000)/APS Outputs/Current Q 3Y0 <-> Data Pointer/QCurrentSetPoints[21]
//     Term 5 (APS4322-7000)/APS Outputs/Current Q 3Y1 <-> Data Pointer/QCurrentSetPoints[22]
//     Term 5 (APS4322-7000)/APS Outputs/Current Q 3Y2 <-> Data Pointer/QCurrentSetPoints[23]
//     Term 5 (APS4322-7000)/APS Outputs/PhiE 0X0 <-> Data Pointer/PhiSetPoints[0]
//     Term 5 (APS4322-7000)/APS Outputs/PhiE 0X1 <-> Data Pointer/PhiSetPoints[1]
//     Term 5 (APS4322-7000)/APS Outputs/PhiE 0X2 <-> Data Pointer/PhiSetPoints[2]
//     Term 5 (APS4322-7000)/APS Outputs/PhiE 1X0 <-> Data Pointer/PhiSetPoints[6]
//     Term 5 (APS4322-7000)/APS Outputs/PhiE 1X1 <-> Data Pointer/PhiSetPoints[7]
//     Term 5 (APS4322-7000)/APS Outputs/PhiE 1X2 <-> Data Pointer/PhiSetPoints[8]
//     Term 5 (APS4322-7000)/APS Outputs/PhiE 2X0 <-> Data Pointer/PhiSetPoints[12]
//     Term 5 (APS4322-7000)/APS Outputs/PhiE 2X1 <-> Data Pointer/PhiSetPoints[13]
//     Term 5 (APS4322-7000)/APS Outputs/PhiE 2X2 <-> Data Pointer/PhiSetPoints[14]
//     Term 5 (APS4322-7000)/APS Outputs/PhiE 3X0 <-> Data Pointer/PhiSetPoints[18]
//     Term 5 (APS4322-7000)/APS Outputs/PhiE 3X1 <-> Data Pointer/PhiSetPoints[19]
//     Term 5 (APS4322-7000)/APS Outputs/PhiE 3X2 <-> Data Pointer/PhiSetPoints[20]
//     Term 5 (APS4322-7000)/APS Outputs/PhiE 0Y0 <-> Data Pointer/PhiSetPoints[3]
//     Term 5 (APS4322-7000)/APS Outputs/PhiE 0Y1 <-> Data Pointer/PhiSetPoints[4]
//     Term 5 (APS4322-7000)/APS Outputs/PhiE 0Y2 <-> Data Pointer/PhiSetPoints[5]
//     Term 5 (APS4322-7000)/APS Outputs/PhiE 1Y0 <-> Data Pointer/PhiSetPoints[9]
//     Term 5 (APS4322-7000)/APS Outputs/PhiE 1Y1 <-> Data Pointer/PhiSetPoints[10]
//     Term 5 (APS4322-7000)/APS Outputs/PhiE 1Y2 <-> Data Pointer/PhiSetPoints[11]
//     Term 5 (APS4322-7000)/APS Outputs/PhiE 2Y0 <-> Data Pointer/PhiSetPoints[15]
//     Term 5 (APS4322-7000)/APS Outputs/PhiE 2Y1 <-> Data Pointer/PhiSetPoints[16]
//     Term 5 (APS4322-7000)/APS Outputs/PhiE 2Y2 <-> Data Pointer/PhiSetPoints[17]
//     Term 5 (APS4322-7000)/APS Outputs/PhiE 3Y0 <-> Data Pointer/PhiSetPoints[21]
//     Term 5 (APS4322-7000)/APS Outputs/PhiE 3Y1 <-> Data Pointer/PhiSetPoints[22]
//     Term 5 (APS4322-7000)/APS Outputs/PhiE 3Y2 <-> Data Pointer/PhiSetPoints[23]
//     Term 5 (APS4322-7000)/Term 6 (APS4322-5000)/FB Inputs/A{0..8 step 2} X-Field <-> Data Pointer/HallSensorFieldsXYZ[{0..12 step 3}]  (5 links)
//     Term 5 (APS4322-7000)/Term 6 (APS4322-5000)/FB Inputs/A{0..8 step 2} Y-Field <-> Data Pointer/HallSensorFieldsXYZ[{1..13 step 3}]  (5 links)
//     Term 5 (APS4322-7000)/Term 6 (APS4322-5000)/FB Inputs/A{0..8 step 2} Z-Field <-> Data Pointer/HallSensorFieldsXYZ[{2..14 step 3}]  (5 links)
//     Term 5 (APS4322-7000)/Term 6 (APS4322-5000)/FB Inputs/B{1..9 step 2} X-Field <-> Data Pointer/HallSensorFieldsXYZ[{15..27 step 3}]  (5 links)
//     Term 5 (APS4322-7000)/Term 6 (APS4322-5000)/FB Inputs/B{1..9 step 2} Y-Field <-> Data Pointer/HallSensorFieldsXYZ[{16..28 step 3}]  (5 links)
//     Term 5 (APS4322-7000)/Term 6 (APS4322-5000)/FB Inputs/B{1..9 step 2} Z-Field <-> Data Pointer/HallSensorFieldsXYZ[{17..29 step 3}]  (5 links)
//     Term 5 (APS4322-7000)/Term 6 (APS4322-5000)/FB Inputs/C{0..8 step 2} X-Field <-> Data Pointer/HallSensorFieldsXYZ[{30..42 step 3}]  (5 links)
//     Term 5 (APS4322-7000)/Term 6 (APS4322-5000)/FB Inputs/C{0..8 step 2} Y-Field <-> Data Pointer/HallSensorFieldsXYZ[{31..43 step 3}]  (5 links)
//     Term 5 (APS4322-7000)/Term 6 (APS4322-5000)/FB Inputs/C{0..8 step 2} Z-Field <-> Data Pointer/HallSensorFieldsXYZ[{32..44 step 3}]  (5 links)
//     Term 5 (APS4322-7000)/Term 6 (APS4322-5000)/FB Inputs/D{1..9 step 2} X-Field <-> Data Pointer/HallSensorFieldsXYZ[{45..57 step 3}]  (5 links)
//     Term 5 (APS4322-7000)/Term 6 (APS4322-5000)/FB Inputs/D{1..9 step 2} Y-Field <-> Data Pointer/HallSensorFieldsXYZ[{46..58 step 3}]  (5 links)
//     Term 5 (APS4322-7000)/Term 6 (APS4322-5000)/FB Inputs/D{1..9 step 2} Z-Field <-> Data Pointer/HallSensorFieldsXYZ[{47..59 step 3}]  (5 links)
//     Term 5 (APS4322-7000)/Term 6 (APS4322-5000)/FB Inputs/E{0..8 step 2} X-Field <-> Data Pointer/HallSensorFieldsXYZ[{60..72 step 3}]  (5 links)
//     Term 5 (APS4322-7000)/Term 6 (APS4322-5000)/FB Inputs/E{0..8 step 2} Y-Field <-> Data Pointer/HallSensorFieldsXYZ[{61..73 step 3}]  (5 links)
//     Term 5 (APS4322-7000)/Term 6 (APS4322-5000)/FB Inputs/E{0..8 step 2} Z-Field <-> Data Pointer/HallSensorFieldsXYZ[{62..74 step 3}]  (5 links)
//     Term 5 (APS4322-7000)/Term 6 (APS4322-5000)/FB Inputs/F{1..9 step 2} X-Field <-> Data Pointer/HallSensorFieldsXYZ[{75..87 step 3}]  (5 links)
//     Term 5 (APS4322-7000)/Term 6 (APS4322-5000)/FB Inputs/F{1..9 step 2} Y-Field <-> Data Pointer/HallSensorFieldsXYZ[{76..88 step 3}]  (5 links)
//     Term 5 (APS4322-7000)/Term 6 (APS4322-5000)/FB Inputs/F{1..9 step 2} Z-Field <-> Data Pointer/HallSensorFieldsXYZ[{77..89 step 3}]  (5 links)
//     Term 5 (APS4322-7000)/Term 6 (APS4322-5000)/FB Inputs/G{0..8 step 2} X-Field <-> Data Pointer/HallSensorFieldsXYZ[{90..102 step 3}]  (5 links)
//     Term 5 (APS4322-7000)/Term 6 (APS4322-5000)/FB Inputs/G{0..8 step 2} Y-Field <-> Data Pointer/HallSensorFieldsXYZ[{91..103 step 3}]  (5 links)
//     Term 5 (APS4322-7000)/Term 6 (APS4322-5000)/FB Inputs/G{0..8 step 2} Z-Field <-> Data Pointer/HallSensorFieldsXYZ[{92..104 step 3}]  (5 links)
//     Term 5 (APS4322-7000)/Term 6 (APS4322-5000)/FB Inputs/H{1..9 step 2} X-Field <-> Data Pointer/HallSensorFieldsXYZ[{105..117 step 3}]  (5 links)
//     Term 5 (APS4322-7000)/Term 6 (APS4322-5000)/FB Inputs/H{1..9 step 2} Y-Field <-> Data Pointer/HallSensorFieldsXYZ[{106..118 step 3}]  (5 links)
//     Term 5 (APS4322-7000)/Term 6 (APS4322-5000)/FB Inputs/H{1..9 step 2} Z-Field <-> Data Pointer/HallSensorFieldsXYZ[{107..119 step 3}]  (5 links)
//     Term 5 (APS4322-7000)/Term 6 (APS4322-5000)/FB Inputs/I{0..8 step 2} X-Field <-> Data Pointer/HallSensorFieldsXYZ[{120..132 step 3}]  (5 links)
//     Term 5 (APS4322-7000)/Term 6 (APS4322-5000)/FB Inputs/I{0..8 step 2} Y-Field <-> Data Pointer/HallSensorFieldsXYZ[{121..133 step 3}]  (5 links)
//     Term 5 (APS4322-7000)/Term 6 (APS4322-5000)/FB Inputs/I{0..8 step 2} Z-Field <-> Data Pointer/HallSensorFieldsXYZ[{122..134 step 3}]  (5 links)
//     Term 5 (APS4322-7000)/Term 6 (APS4322-5000)/FB Inputs/J{1..9 step 2} X-Field <-> Data Pointer/HallSensorFieldsXYZ[{135..147 step 3}]  (5 links)
//     Term 5 (APS4322-7000)/Term 6 (APS4322-5000)/FB Inputs/J{1..9 step 2} Y-Field <-> Data Pointer/HallSensorFieldsXYZ[{136..148 step 3}]  (5 links)
//     Term 5 (APS4322-7000)/Term 6 (APS4322-5000)/FB Inputs/J{1..9 step 2} Z-Field <-> Data Pointer/HallSensorFieldsXYZ[{137..149 step 3}]  (5 links)
//     Term 5 (APS4322-7000)/Term 6 (APS4322-5000)/FB Inputs/Status <-> Data Pointer/FeedbackStatus
//   Device 2 (EtherCAT) <-> TcCOM Objects/XPlanar/Part1/APS4322_P1_4
//     Term 7 (APS4322-7000)/APS Comm Inputs/CommStatusWord <-> Data Pointer/MoverCommStatusWord
//     Term 7 (APS4322-7000)/APS Comm Inputs/Data {1..4} <-> Data Pointer/MoverCommDataIn[{0..3}]  (4 links)
//     Term 7 (APS4322-7000)/APS Comm Outputs/CommControlWord <-> Data Pointer/MoverCommControlWord
//     Term 7 (APS4322-7000)/APS Comm Outputs/Data 1 <-> Data Pointer/MoverCommDataOut
//     Term 7 (APS4322-7000)/APS Diagdata/DC Link Voltage <-> Data Pointer/DcLinkVoltage
//     Term 7 (APS4322-7000)/APS Diagdata/Power supply current <-> Data Pointer/PowerSupplyCurrent
//     Term 7 (APS4322-7000)/APS Inputs/StatusWord <-> Data Pointer/PowerUnitStatusWord
//     Term 7 (APS4322-7000)/APS Outputs/ControlWord <-> Data Pointer/PowerUnitControlWord
//     Term 7 (APS4322-7000)/APS Outputs/Current D 0X0 <-> Data Pointer/DCurrentSetPoints[0]
//     Term 7 (APS4322-7000)/APS Outputs/Current D 0X1 <-> Data Pointer/DCurrentSetPoints[1]
//     Term 7 (APS4322-7000)/APS Outputs/Current D 0X2 <-> Data Pointer/DCurrentSetPoints[2]
//     Term 7 (APS4322-7000)/APS Outputs/Current D 1X0 <-> Data Pointer/DCurrentSetPoints[6]
//     Term 7 (APS4322-7000)/APS Outputs/Current D 1X1 <-> Data Pointer/DCurrentSetPoints[7]
//     Term 7 (APS4322-7000)/APS Outputs/Current D 1X2 <-> Data Pointer/DCurrentSetPoints[8]
//     Term 7 (APS4322-7000)/APS Outputs/Current D 2X0 <-> Data Pointer/DCurrentSetPoints[12]
//     Term 7 (APS4322-7000)/APS Outputs/Current D 2X1 <-> Data Pointer/DCurrentSetPoints[13]
//     Term 7 (APS4322-7000)/APS Outputs/Current D 2X2 <-> Data Pointer/DCurrentSetPoints[14]
//     Term 7 (APS4322-7000)/APS Outputs/Current D 3X0 <-> Data Pointer/DCurrentSetPoints[18]
//     Term 7 (APS4322-7000)/APS Outputs/Current D 3X1 <-> Data Pointer/DCurrentSetPoints[19]
//     Term 7 (APS4322-7000)/APS Outputs/Current D 3X2 <-> Data Pointer/DCurrentSetPoints[20]
//     Term 7 (APS4322-7000)/APS Outputs/Current D 0Y0 <-> Data Pointer/DCurrentSetPoints[3]
//     Term 7 (APS4322-7000)/APS Outputs/Current D 0Y1 <-> Data Pointer/DCurrentSetPoints[4]
//     Term 7 (APS4322-7000)/APS Outputs/Current D 0Y2 <-> Data Pointer/DCurrentSetPoints[5]
//     Term 7 (APS4322-7000)/APS Outputs/Current D 1Y0 <-> Data Pointer/DCurrentSetPoints[9]
//     Term 7 (APS4322-7000)/APS Outputs/Current D 1Y1 <-> Data Pointer/DCurrentSetPoints[10]
//     Term 7 (APS4322-7000)/APS Outputs/Current D 1Y2 <-> Data Pointer/DCurrentSetPoints[11]
//     Term 7 (APS4322-7000)/APS Outputs/Current D 2Y0 <-> Data Pointer/DCurrentSetPoints[15]
//     Term 7 (APS4322-7000)/APS Outputs/Current D 2Y1 <-> Data Pointer/DCurrentSetPoints[16]
//     Term 7 (APS4322-7000)/APS Outputs/Current D 2Y2 <-> Data Pointer/DCurrentSetPoints[17]
//     Term 7 (APS4322-7000)/APS Outputs/Current D 3Y0 <-> Data Pointer/DCurrentSetPoints[21]
//     Term 7 (APS4322-7000)/APS Outputs/Current D 3Y1 <-> Data Pointer/DCurrentSetPoints[22]
//     Term 7 (APS4322-7000)/APS Outputs/Current D 3Y2 <-> Data Pointer/DCurrentSetPoints[23]
//     Term 7 (APS4322-7000)/APS Outputs/Current Q 0X0 <-> Data Pointer/QCurrentSetPoints[0]
//     Term 7 (APS4322-7000)/APS Outputs/Current Q 0X1 <-> Data Pointer/QCurrentSetPoints[1]
//     Term 7 (APS4322-7000)/APS Outputs/Current Q 0X2 <-> Data Pointer/QCurrentSetPoints[2]
//     Term 7 (APS4322-7000)/APS Outputs/Current Q 1X0 <-> Data Pointer/QCurrentSetPoints[6]
//     Term 7 (APS4322-7000)/APS Outputs/Current Q 1X1 <-> Data Pointer/QCurrentSetPoints[7]
//     Term 7 (APS4322-7000)/APS Outputs/Current Q 1X2 <-> Data Pointer/QCurrentSetPoints[8]
//     Term 7 (APS4322-7000)/APS Outputs/Current Q 2X0 <-> Data Pointer/QCurrentSetPoints[12]
//     Term 7 (APS4322-7000)/APS Outputs/Current Q 2X1 <-> Data Pointer/QCurrentSetPoints[13]
//     Term 7 (APS4322-7000)/APS Outputs/Current Q 2X2 <-> Data Pointer/QCurrentSetPoints[14]
//     Term 7 (APS4322-7000)/APS Outputs/Current Q 3X0 <-> Data Pointer/QCurrentSetPoints[18]
//     Term 7 (APS4322-7000)/APS Outputs/Current Q 3X1 <-> Data Pointer/QCurrentSetPoints[19]
//     Term 7 (APS4322-7000)/APS Outputs/Current Q 3X2 <-> Data Pointer/QCurrentSetPoints[20]
//     Term 7 (APS4322-7000)/APS Outputs/Current Q 0Y0 <-> Data Pointer/QCurrentSetPoints[3]
//     Term 7 (APS4322-7000)/APS Outputs/Current Q 0Y1 <-> Data Pointer/QCurrentSetPoints[4]
//     Term 7 (APS4322-7000)/APS Outputs/Current Q 0Y2 <-> Data Pointer/QCurrentSetPoints[5]
//     Term 7 (APS4322-7000)/APS Outputs/Current Q 1Y0 <-> Data Pointer/QCurrentSetPoints[9]
//     Term 7 (APS4322-7000)/APS Outputs/Current Q 1Y1 <-> Data Pointer/QCurrentSetPoints[10]
//     Term 7 (APS4322-7000)/APS Outputs/Current Q 1Y2 <-> Data Pointer/QCurrentSetPoints[11]
//     Term 7 (APS4322-7000)/APS Outputs/Current Q 2Y0 <-> Data Pointer/QCurrentSetPoints[15]
//     Term 7 (APS4322-7000)/APS Outputs/Current Q 2Y1 <-> Data Pointer/QCurrentSetPoints[16]
//     Term 7 (APS4322-7000)/APS Outputs/Current Q 2Y2 <-> Data Pointer/QCurrentSetPoints[17]
//     Term 7 (APS4322-7000)/APS Outputs/Current Q 3Y0 <-> Data Pointer/QCurrentSetPoints[21]
//     Term 7 (APS4322-7000)/APS Outputs/Current Q 3Y1 <-> Data Pointer/QCurrentSetPoints[22]
//     Term 7 (APS4322-7000)/APS Outputs/Current Q 3Y2 <-> Data Pointer/QCurrentSetPoints[23]
//     Term 7 (APS4322-7000)/APS Outputs/PhiE 0X0 <-> Data Pointer/PhiSetPoints[0]
//     Term 7 (APS4322-7000)/APS Outputs/PhiE 0X1 <-> Data Pointer/PhiSetPoints[1]
//     Term 7 (APS4322-7000)/APS Outputs/PhiE 0X2 <-> Data Pointer/PhiSetPoints[2]
//     Term 7 (APS4322-7000)/APS Outputs/PhiE 1X0 <-> Data Pointer/PhiSetPoints[6]
//     Term 7 (APS4322-7000)/APS Outputs/PhiE 1X1 <-> Data Pointer/PhiSetPoints[7]
//     Term 7 (APS4322-7000)/APS Outputs/PhiE 1X2 <-> Data Pointer/PhiSetPoints[8]
//     Term 7 (APS4322-7000)/APS Outputs/PhiE 2X0 <-> Data Pointer/PhiSetPoints[12]
//     Term 7 (APS4322-7000)/APS Outputs/PhiE 2X1 <-> Data Pointer/PhiSetPoints[13]
//     Term 7 (APS4322-7000)/APS Outputs/PhiE 2X2 <-> Data Pointer/PhiSetPoints[14]
//     Term 7 (APS4322-7000)/APS Outputs/PhiE 3X0 <-> Data Pointer/PhiSetPoints[18]
//     Term 7 (APS4322-7000)/APS Outputs/PhiE 3X1 <-> Data Pointer/PhiSetPoints[19]
//     Term 7 (APS4322-7000)/APS Outputs/PhiE 3X2 <-> Data Pointer/PhiSetPoints[20]
//     Term 7 (APS4322-7000)/APS Outputs/PhiE 0Y0 <-> Data Pointer/PhiSetPoints[3]
//     Term 7 (APS4322-7000)/APS Outputs/PhiE 0Y1 <-> Data Pointer/PhiSetPoints[4]
//     Term 7 (APS4322-7000)/APS Outputs/PhiE 0Y2 <-> Data Pointer/PhiSetPoints[5]
//     Term 7 (APS4322-7000)/APS Outputs/PhiE 1Y0 <-> Data Pointer/PhiSetPoints[9]
//     Term 7 (APS4322-7000)/APS Outputs/PhiE 1Y1 <-> Data Pointer/PhiSetPoints[10]
//     Term 7 (APS4322-7000)/APS Outputs/PhiE 1Y2 <-> Data Pointer/PhiSetPoints[11]
//     Term 7 (APS4322-7000)/APS Outputs/PhiE 2Y0 <-> Data Pointer/PhiSetPoints[15]
//     Term 7 (APS4322-7000)/APS Outputs/PhiE 2Y1 <-> Data Pointer/PhiSetPoints[16]
//     Term 7 (APS4322-7000)/APS Outputs/PhiE 2Y2 <-> Data Pointer/PhiSetPoints[17]
//     Term 7 (APS4322-7000)/APS Outputs/PhiE 3Y0 <-> Data Pointer/PhiSetPoints[21]
//     Term 7 (APS4322-7000)/APS Outputs/PhiE 3Y1 <-> Data Pointer/PhiSetPoints[22]
//     Term 7 (APS4322-7000)/APS Outputs/PhiE 3Y2 <-> Data Pointer/PhiSetPoints[23]
//     Term 7 (APS4322-7000)/Term 8 (APS4322-5000)/FB Inputs/A{0..8 step 2} X-Field <-> Data Pointer/HallSensorFieldsXYZ[{0..12 step 3}]  (5 links)
//     Term 7 (APS4322-7000)/Term 8 (APS4322-5000)/FB Inputs/A{0..8 step 2} Y-Field <-> Data Pointer/HallSensorFieldsXYZ[{1..13 step 3}]  (5 links)
//     Term 7 (APS4322-7000)/Term 8 (APS4322-5000)/FB Inputs/A{0..8 step 2} Z-Field <-> Data Pointer/HallSensorFieldsXYZ[{2..14 step 3}]  (5 links)
//     Term 7 (APS4322-7000)/Term 8 (APS4322-5000)/FB Inputs/B{1..9 step 2} X-Field <-> Data Pointer/HallSensorFieldsXYZ[{15..27 step 3}]  (5 links)
//     Term 7 (APS4322-7000)/Term 8 (APS4322-5000)/FB Inputs/B{1..9 step 2} Y-Field <-> Data Pointer/HallSensorFieldsXYZ[{16..28 step 3}]  (5 links)
//     Term 7 (APS4322-7000)/Term 8 (APS4322-5000)/FB Inputs/B{1..9 step 2} Z-Field <-> Data Pointer/HallSensorFieldsXYZ[{17..29 step 3}]  (5 links)
//     Term 7 (APS4322-7000)/Term 8 (APS4322-5000)/FB Inputs/C{0..8 step 2} X-Field <-> Data Pointer/HallSensorFieldsXYZ[{30..42 step 3}]  (5 links)
//     Term 7 (APS4322-7000)/Term 8 (APS4322-5000)/FB Inputs/C{0..8 step 2} Y-Field <-> Data Pointer/HallSensorFieldsXYZ[{31..43 step 3}]  (5 links)
//     Term 7 (APS4322-7000)/Term 8 (APS4322-5000)/FB Inputs/C{0..8 step 2} Z-Field <-> Data Pointer/HallSensorFieldsXYZ[{32..44 step 3}]  (5 links)
//     Term 7 (APS4322-7000)/Term 8 (APS4322-5000)/FB Inputs/D{1..9 step 2} X-Field <-> Data Pointer/HallSensorFieldsXYZ[{45..57 step 3}]  (5 links)
//     Term 7 (APS4322-7000)/Term 8 (APS4322-5000)/FB Inputs/D{1..9 step 2} Y-Field <-> Data Pointer/HallSensorFieldsXYZ[{46..58 step 3}]  (5 links)
//     Term 7 (APS4322-7000)/Term 8 (APS4322-5000)/FB Inputs/D{1..9 step 2} Z-Field <-> Data Pointer/HallSensorFieldsXYZ[{47..59 step 3}]  (5 links)
//     Term 7 (APS4322-7000)/Term 8 (APS4322-5000)/FB Inputs/E{0..8 step 2} X-Field <-> Data Pointer/HallSensorFieldsXYZ[{60..72 step 3}]  (5 links)
//     Term 7 (APS4322-7000)/Term 8 (APS4322-5000)/FB Inputs/E{0..8 step 2} Y-Field <-> Data Pointer/HallSensorFieldsXYZ[{61..73 step 3}]  (5 links)
//     Term 7 (APS4322-7000)/Term 8 (APS4322-5000)/FB Inputs/E{0..8 step 2} Z-Field <-> Data Pointer/HallSensorFieldsXYZ[{62..74 step 3}]  (5 links)
//     Term 7 (APS4322-7000)/Term 8 (APS4322-5000)/FB Inputs/F{1..9 step 2} X-Field <-> Data Pointer/HallSensorFieldsXYZ[{75..87 step 3}]  (5 links)
//     Term 7 (APS4322-7000)/Term 8 (APS4322-5000)/FB Inputs/F{1..9 step 2} Y-Field <-> Data Pointer/HallSensorFieldsXYZ[{76..88 step 3}]  (5 links)
//     Term 7 (APS4322-7000)/Term 8 (APS4322-5000)/FB Inputs/F{1..9 step 2} Z-Field <-> Data Pointer/HallSensorFieldsXYZ[{77..89 step 3}]  (5 links)
//     Term 7 (APS4322-7000)/Term 8 (APS4322-5000)/FB Inputs/G{0..8 step 2} X-Field <-> Data Pointer/HallSensorFieldsXYZ[{90..102 step 3}]  (5 links)
//     Term 7 (APS4322-7000)/Term 8 (APS4322-5000)/FB Inputs/G{0..8 step 2} Y-Field <-> Data Pointer/HallSensorFieldsXYZ[{91..103 step 3}]  (5 links)
//     Term 7 (APS4322-7000)/Term 8 (APS4322-5000)/FB Inputs/G{0..8 step 2} Z-Field <-> Data Pointer/HallSensorFieldsXYZ[{92..104 step 3}]  (5 links)
//     Term 7 (APS4322-7000)/Term 8 (APS4322-5000)/FB Inputs/H{1..9 step 2} X-Field <-> Data Pointer/HallSensorFieldsXYZ[{105..117 step 3}]  (5 links)
//     Term 7 (APS4322-7000)/Term 8 (APS4322-5000)/FB Inputs/H{1..9 step 2} Y-Field <-> Data Pointer/HallSensorFieldsXYZ[{106..118 step 3}]  (5 links)
//     Term 7 (APS4322-7000)/Term 8 (APS4322-5000)/FB Inputs/H{1..9 step 2} Z-Field <-> Data Pointer/HallSensorFieldsXYZ[{107..119 step 3}]  (5 links)
//     Term 7 (APS4322-7000)/Term 8 (APS4322-5000)/FB Inputs/I{0..8 step 2} X-Field <-> Data Pointer/HallSensorFieldsXYZ[{120..132 step 3}]  (5 links)
//     Term 7 (APS4322-7000)/Term 8 (APS4322-5000)/FB Inputs/I{0..8 step 2} Y-Field <-> Data Pointer/HallSensorFieldsXYZ[{121..133 step 3}]  (5 links)
//     Term 7 (APS4322-7000)/Term 8 (APS4322-5000)/FB Inputs/I{0..8 step 2} Z-Field <-> Data Pointer/HallSensorFieldsXYZ[{122..134 step 3}]  (5 links)
//     Term 7 (APS4322-7000)/Term 8 (APS4322-5000)/FB Inputs/J{1..9 step 2} X-Field <-> Data Pointer/HallSensorFieldsXYZ[{135..147 step 3}]  (5 links)
//     Term 7 (APS4322-7000)/Term 8 (APS4322-5000)/FB Inputs/J{1..9 step 2} Y-Field <-> Data Pointer/HallSensorFieldsXYZ[{136..148 step 3}]  (5 links)
//     Term 7 (APS4322-7000)/Term 8 (APS4322-5000)/FB Inputs/J{1..9 step 2} Z-Field <-> Data Pointer/HallSensorFieldsXYZ[{137..149 step 3}]  (5 links)
//     Term 7 (APS4322-7000)/Term 8 (APS4322-5000)/FB Inputs/Status <-> Data Pointer/FeedbackStatus
//   Device 2 (EtherCAT) <-> TcCOM Objects/XPlanar/Part1/APS4322_P1_5
//     Term 9 (APS4322-7000)/APS Comm Inputs/CommStatusWord <-> Data Pointer/MoverCommStatusWord
//     Term 9 (APS4322-7000)/APS Comm Inputs/Data {1..4} <-> Data Pointer/MoverCommDataIn[{0..3}]  (4 links)
//     Term 9 (APS4322-7000)/APS Comm Outputs/CommControlWord <-> Data Pointer/MoverCommControlWord
//     Term 9 (APS4322-7000)/APS Comm Outputs/Data 1 <-> Data Pointer/MoverCommDataOut
//     Term 9 (APS4322-7000)/APS Diagdata/DC Link Voltage <-> Data Pointer/DcLinkVoltage
//     Term 9 (APS4322-7000)/APS Diagdata/Power supply current <-> Data Pointer/PowerSupplyCurrent
//     Term 9 (APS4322-7000)/APS Inputs/StatusWord <-> Data Pointer/PowerUnitStatusWord
//     Term 9 (APS4322-7000)/APS Outputs/ControlWord <-> Data Pointer/PowerUnitControlWord
//     Term 9 (APS4322-7000)/APS Outputs/Current D 0X0 <-> Data Pointer/DCurrentSetPoints[0]
//     Term 9 (APS4322-7000)/APS Outputs/Current D 0X1 <-> Data Pointer/DCurrentSetPoints[1]
//     Term 9 (APS4322-7000)/APS Outputs/Current D 0X2 <-> Data Pointer/DCurrentSetPoints[2]
//     Term 9 (APS4322-7000)/APS Outputs/Current D 1X0 <-> Data Pointer/DCurrentSetPoints[6]
//     Term 9 (APS4322-7000)/APS Outputs/Current D 1X1 <-> Data Pointer/DCurrentSetPoints[7]
//     Term 9 (APS4322-7000)/APS Outputs/Current D 1X2 <-> Data Pointer/DCurrentSetPoints[8]
//     Term 9 (APS4322-7000)/APS Outputs/Current D 2X0 <-> Data Pointer/DCurrentSetPoints[12]
//     Term 9 (APS4322-7000)/APS Outputs/Current D 2X1 <-> Data Pointer/DCurrentSetPoints[13]
//     Term 9 (APS4322-7000)/APS Outputs/Current D 2X2 <-> Data Pointer/DCurrentSetPoints[14]
//     Term 9 (APS4322-7000)/APS Outputs/Current D 3X0 <-> Data Pointer/DCurrentSetPoints[18]
//     Term 9 (APS4322-7000)/APS Outputs/Current D 3X1 <-> Data Pointer/DCurrentSetPoints[19]
//     Term 9 (APS4322-7000)/APS Outputs/Current D 3X2 <-> Data Pointer/DCurrentSetPoints[20]
//     Term 9 (APS4322-7000)/APS Outputs/Current D 0Y0 <-> Data Pointer/DCurrentSetPoints[3]
//     Term 9 (APS4322-7000)/APS Outputs/Current D 0Y1 <-> Data Pointer/DCurrentSetPoints[4]
//     Term 9 (APS4322-7000)/APS Outputs/Current D 0Y2 <-> Data Pointer/DCurrentSetPoints[5]
//     Term 9 (APS4322-7000)/APS Outputs/Current D 1Y0 <-> Data Pointer/DCurrentSetPoints[9]
//     Term 9 (APS4322-7000)/APS Outputs/Current D 1Y1 <-> Data Pointer/DCurrentSetPoints[10]
//     Term 9 (APS4322-7000)/APS Outputs/Current D 1Y2 <-> Data Pointer/DCurrentSetPoints[11]
//     Term 9 (APS4322-7000)/APS Outputs/Current D 2Y0 <-> Data Pointer/DCurrentSetPoints[15]
//     Term 9 (APS4322-7000)/APS Outputs/Current D 2Y1 <-> Data Pointer/DCurrentSetPoints[16]
//     Term 9 (APS4322-7000)/APS Outputs/Current D 2Y2 <-> Data Pointer/DCurrentSetPoints[17]
//     Term 9 (APS4322-7000)/APS Outputs/Current D 3Y0 <-> Data Pointer/DCurrentSetPoints[21]
//     Term 9 (APS4322-7000)/APS Outputs/Current D 3Y1 <-> Data Pointer/DCurrentSetPoints[22]
//     Term 9 (APS4322-7000)/APS Outputs/Current D 3Y2 <-> Data Pointer/DCurrentSetPoints[23]
//     Term 9 (APS4322-7000)/APS Outputs/Current Q 0X0 <-> Data Pointer/QCurrentSetPoints[0]
//     Term 9 (APS4322-7000)/APS Outputs/Current Q 0X1 <-> Data Pointer/QCurrentSetPoints[1]
//     Term 9 (APS4322-7000)/APS Outputs/Current Q 0X2 <-> Data Pointer/QCurrentSetPoints[2]
//     Term 9 (APS4322-7000)/APS Outputs/Current Q 1X0 <-> Data Pointer/QCurrentSetPoints[6]
//     Term 9 (APS4322-7000)/APS Outputs/Current Q 1X1 <-> Data Pointer/QCurrentSetPoints[7]
//     Term 9 (APS4322-7000)/APS Outputs/Current Q 1X2 <-> Data Pointer/QCurrentSetPoints[8]
//     Term 9 (APS4322-7000)/APS Outputs/Current Q 2X0 <-> Data Pointer/QCurrentSetPoints[12]
//     Term 9 (APS4322-7000)/APS Outputs/Current Q 2X1 <-> Data Pointer/QCurrentSetPoints[13]
//     Term 9 (APS4322-7000)/APS Outputs/Current Q 2X2 <-> Data Pointer/QCurrentSetPoints[14]
//     Term 9 (APS4322-7000)/APS Outputs/Current Q 3X0 <-> Data Pointer/QCurrentSetPoints[18]
//     Term 9 (APS4322-7000)/APS Outputs/Current Q 3X1 <-> Data Pointer/QCurrentSetPoints[19]
//     Term 9 (APS4322-7000)/APS Outputs/Current Q 3X2 <-> Data Pointer/QCurrentSetPoints[20]
//     Term 9 (APS4322-7000)/APS Outputs/Current Q 0Y0 <-> Data Pointer/QCurrentSetPoints[3]
//     Term 9 (APS4322-7000)/APS Outputs/Current Q 0Y1 <-> Data Pointer/QCurrentSetPoints[4]
//     Term 9 (APS4322-7000)/APS Outputs/Current Q 0Y2 <-> Data Pointer/QCurrentSetPoints[5]
//     Term 9 (APS4322-7000)/APS Outputs/Current Q 1Y0 <-> Data Pointer/QCurrentSetPoints[9]
//     Term 9 (APS4322-7000)/APS Outputs/Current Q 1Y1 <-> Data Pointer/QCurrentSetPoints[10]
//     Term 9 (APS4322-7000)/APS Outputs/Current Q 1Y2 <-> Data Pointer/QCurrentSetPoints[11]
//     Term 9 (APS4322-7000)/APS Outputs/Current Q 2Y0 <-> Data Pointer/QCurrentSetPoints[15]
//     Term 9 (APS4322-7000)/APS Outputs/Current Q 2Y1 <-> Data Pointer/QCurrentSetPoints[16]
//     Term 9 (APS4322-7000)/APS Outputs/Current Q 2Y2 <-> Data Pointer/QCurrentSetPoints[17]
//     Term 9 (APS4322-7000)/APS Outputs/Current Q 3Y0 <-> Data Pointer/QCurrentSetPoints[21]
//     Term 9 (APS4322-7000)/APS Outputs/Current Q 3Y1 <-> Data Pointer/QCurrentSetPoints[22]
//     Term 9 (APS4322-7000)/APS Outputs/Current Q 3Y2 <-> Data Pointer/QCurrentSetPoints[23]
//     Term 9 (APS4322-7000)/APS Outputs/PhiE 0X0 <-> Data Pointer/PhiSetPoints[0]
//     Term 9 (APS4322-7000)/APS Outputs/PhiE 0X1 <-> Data Pointer/PhiSetPoints[1]
//     Term 9 (APS4322-7000)/APS Outputs/PhiE 0X2 <-> Data Pointer/PhiSetPoints[2]
//     Term 9 (APS4322-7000)/APS Outputs/PhiE 1X0 <-> Data Pointer/PhiSetPoints[6]
//     Term 9 (APS4322-7000)/APS Outputs/PhiE 1X1 <-> Data Pointer/PhiSetPoints[7]
//     Term 9 (APS4322-7000)/APS Outputs/PhiE 1X2 <-> Data Pointer/PhiSetPoints[8]
//     Term 9 (APS4322-7000)/APS Outputs/PhiE 2X0 <-> Data Pointer/PhiSetPoints[12]
//     Term 9 (APS4322-7000)/APS Outputs/PhiE 2X1 <-> Data Pointer/PhiSetPoints[13]
//     Term 9 (APS4322-7000)/APS Outputs/PhiE 2X2 <-> Data Pointer/PhiSetPoints[14]
//     Term 9 (APS4322-7000)/APS Outputs/PhiE 3X0 <-> Data Pointer/PhiSetPoints[18]
//     Term 9 (APS4322-7000)/APS Outputs/PhiE 3X1 <-> Data Pointer/PhiSetPoints[19]
//     Term 9 (APS4322-7000)/APS Outputs/PhiE 3X2 <-> Data Pointer/PhiSetPoints[20]
//     Term 9 (APS4322-7000)/APS Outputs/PhiE 0Y0 <-> Data Pointer/PhiSetPoints[3]
//     Term 9 (APS4322-7000)/APS Outputs/PhiE 0Y1 <-> Data Pointer/PhiSetPoints[4]
//     Term 9 (APS4322-7000)/APS Outputs/PhiE 0Y2 <-> Data Pointer/PhiSetPoints[5]
//     Term 9 (APS4322-7000)/APS Outputs/PhiE 1Y0 <-> Data Pointer/PhiSetPoints[9]
//     Term 9 (APS4322-7000)/APS Outputs/PhiE 1Y1 <-> Data Pointer/PhiSetPoints[10]
//     Term 9 (APS4322-7000)/APS Outputs/PhiE 1Y2 <-> Data Pointer/PhiSetPoints[11]
//     Term 9 (APS4322-7000)/APS Outputs/PhiE 2Y0 <-> Data Pointer/PhiSetPoints[15]
//     Term 9 (APS4322-7000)/APS Outputs/PhiE 2Y1 <-> Data Pointer/PhiSetPoints[16]
//     Term 9 (APS4322-7000)/APS Outputs/PhiE 2Y2 <-> Data Pointer/PhiSetPoints[17]
//     Term 9 (APS4322-7000)/APS Outputs/PhiE 3Y0 <-> Data Pointer/PhiSetPoints[21]
//     Term 9 (APS4322-7000)/APS Outputs/PhiE 3Y1 <-> Data Pointer/PhiSetPoints[22]
//     Term 9 (APS4322-7000)/APS Outputs/PhiE 3Y2 <-> Data Pointer/PhiSetPoints[23]
//     Term 9 (APS4322-7000)/Term 10 (APS4322-5000)/FB Inputs/A{0..8 step 2} X-Field <-> Data Pointer/HallSensorFieldsXYZ[{0..12 step 3}]  (5 links)
//     Term 9 (APS4322-7000)/Term 10 (APS4322-5000)/FB Inputs/A{0..8 step 2} Y-Field <-> Data Pointer/HallSensorFieldsXYZ[{1..13 step 3}]  (5 links)
//     Term 9 (APS4322-7000)/Term 10 (APS4322-5000)/FB Inputs/A{0..8 step 2} Z-Field <-> Data Pointer/HallSensorFieldsXYZ[{2..14 step 3}]  (5 links)
//     Term 9 (APS4322-7000)/Term 10 (APS4322-5000)/FB Inputs/B{1..9 step 2} X-Field <-> Data Pointer/HallSensorFieldsXYZ[{15..27 step 3}]  (5 links)
//     Term 9 (APS4322-7000)/Term 10 (APS4322-5000)/FB Inputs/B{1..9 step 2} Y-Field <-> Data Pointer/HallSensorFieldsXYZ[{16..28 step 3}]  (5 links)
//     Term 9 (APS4322-7000)/Term 10 (APS4322-5000)/FB Inputs/B{1..9 step 2} Z-Field <-> Data Pointer/HallSensorFieldsXYZ[{17..29 step 3}]  (5 links)
//     Term 9 (APS4322-7000)/Term 10 (APS4322-5000)/FB Inputs/C{0..8 step 2} X-Field <-> Data Pointer/HallSensorFieldsXYZ[{30..42 step 3}]  (5 links)
//     Term 9 (APS4322-7000)/Term 10 (APS4322-5000)/FB Inputs/C{0..8 step 2} Y-Field <-> Data Pointer/HallSensorFieldsXYZ[{31..43 step 3}]  (5 links)
//     Term 9 (APS4322-7000)/Term 10 (APS4322-5000)/FB Inputs/C{0..8 step 2} Z-Field <-> Data Pointer/HallSensorFieldsXYZ[{32..44 step 3}]  (5 links)
//     Term 9 (APS4322-7000)/Term 10 (APS4322-5000)/FB Inputs/D{1..9 step 2} X-Field <-> Data Pointer/HallSensorFieldsXYZ[{45..57 step 3}]  (5 links)
//     Term 9 (APS4322-7000)/Term 10 (APS4322-5000)/FB Inputs/D{1..9 step 2} Y-Field <-> Data Pointer/HallSensorFieldsXYZ[{46..58 step 3}]  (5 links)
//     Term 9 (APS4322-7000)/Term 10 (APS4322-5000)/FB Inputs/D{1..9 step 2} Z-Field <-> Data Pointer/HallSensorFieldsXYZ[{47..59 step 3}]  (5 links)
//     Term 9 (APS4322-7000)/Term 10 (APS4322-5000)/FB Inputs/E{0..8 step 2} X-Field <-> Data Pointer/HallSensorFieldsXYZ[{60..72 step 3}]  (5 links)
//     Term 9 (APS4322-7000)/Term 10 (APS4322-5000)/FB Inputs/E{0..8 step 2} Y-Field <-> Data Pointer/HallSensorFieldsXYZ[{61..73 step 3}]  (5 links)
//     Term 9 (APS4322-7000)/Term 10 (APS4322-5000)/FB Inputs/E{0..8 step 2} Z-Field <-> Data Pointer/HallSensorFieldsXYZ[{62..74 step 3}]  (5 links)
//     Term 9 (APS4322-7000)/Term 10 (APS4322-5000)/FB Inputs/F{1..9 step 2} X-Field <-> Data Pointer/HallSensorFieldsXYZ[{75..87 step 3}]  (5 links)
//     Term 9 (APS4322-7000)/Term 10 (APS4322-5000)/FB Inputs/F{1..9 step 2} Y-Field <-> Data Pointer/HallSensorFieldsXYZ[{76..88 step 3}]  (5 links)
//     Term 9 (APS4322-7000)/Term 10 (APS4322-5000)/FB Inputs/F{1..9 step 2} Z-Field <-> Data Pointer/HallSensorFieldsXYZ[{77..89 step 3}]  (5 links)
//     Term 9 (APS4322-7000)/Term 10 (APS4322-5000)/FB Inputs/G{0..8 step 2} X-Field <-> Data Pointer/HallSensorFieldsXYZ[{90..102 step 3}]  (5 links)
//     Term 9 (APS4322-7000)/Term 10 (APS4322-5000)/FB Inputs/G{0..8 step 2} Y-Field <-> Data Pointer/HallSensorFieldsXYZ[{91..103 step 3}]  (5 links)
//     Term 9 (APS4322-7000)/Term 10 (APS4322-5000)/FB Inputs/G{0..8 step 2} Z-Field <-> Data Pointer/HallSensorFieldsXYZ[{92..104 step 3}]  (5 links)
//     Term 9 (APS4322-7000)/Term 10 (APS4322-5000)/FB Inputs/H{1..9 step 2} X-Field <-> Data Pointer/HallSensorFieldsXYZ[{105..117 step 3}]  (5 links)
//     Term 9 (APS4322-7000)/Term 10 (APS4322-5000)/FB Inputs/H{1..9 step 2} Y-Field <-> Data Pointer/HallSensorFieldsXYZ[{106..118 step 3}]  (5 links)
//     Term 9 (APS4322-7000)/Term 10 (APS4322-5000)/FB Inputs/H{1..9 step 2} Z-Field <-> Data Pointer/HallSensorFieldsXYZ[{107..119 step 3}]  (5 links)
//     Term 9 (APS4322-7000)/Term 10 (APS4322-5000)/FB Inputs/I{0..8 step 2} X-Field <-> Data Pointer/HallSensorFieldsXYZ[{120..132 step 3}]  (5 links)
//     Term 9 (APS4322-7000)/Term 10 (APS4322-5000)/FB Inputs/I{0..8 step 2} Y-Field <-> Data Pointer/HallSensorFieldsXYZ[{121..133 step 3}]  (5 links)
//     Term 9 (APS4322-7000)/Term 10 (APS4322-5000)/FB Inputs/I{0..8 step 2} Z-Field <-> Data Pointer/HallSensorFieldsXYZ[{122..134 step 3}]  (5 links)
//     Term 9 (APS4322-7000)/Term 10 (APS4322-5000)/FB Inputs/J{1..9 step 2} X-Field <-> Data Pointer/HallSensorFieldsXYZ[{135..147 step 3}]  (5 links)
//     Term 9 (APS4322-7000)/Term 10 (APS4322-5000)/FB Inputs/J{1..9 step 2} Y-Field <-> Data Pointer/HallSensorFieldsXYZ[{136..148 step 3}]  (5 links)
//     Term 9 (APS4322-7000)/Term 10 (APS4322-5000)/FB Inputs/J{1..9 step 2} Z-Field <-> Data Pointer/HallSensorFieldsXYZ[{137..149 step 3}]  (5 links)
//     Term 9 (APS4322-7000)/Term 10 (APS4322-5000)/FB Inputs/Status <-> Data Pointer/FeedbackStatus
//   XPlanar MC Project/Axes/0000lckx <-> TcCOM Objects/XPlanar/0000lckx
//     IoToMc/STD <-> OutputsToNC3/HWToNC3
//     McToIo/STD <-> InputsFromNC3/NC3ToHW
//   XPlanar MC Project/Axes/0000lcle <-> TcCOM Objects/XPlanar/0000lcle
//     IoToMc/STD <-> OutputsToNC3/HWToNC3
//     McToIo/STD <-> InputsFromNC3/NC3ToHW
//   DMMS_PLC/DMMS_PLC Instance <-> XPlanar MC Project/Axes/0000lckx
//     PlcTask Inputs/MAIN.fbXMotionUnit.fbXPlanarMover[1].stMoverRef.MCTOPLC/ACT <-> McToPlc/ACT
//     PlcTask Inputs/MAIN.fbXMotionUnit.fbXPlanarMover[1].stMoverRef.MCTOPLC/COORDMODE <-> McToPlc/COORDMODE
//     PlcTask Inputs/MAIN.fbXMotionUnit.fbXPlanarMover[1].stMoverRef.MCTOPLC/SET <-> McToPlc/SET
//     PlcTask Inputs/MAIN.fbXMotionUnit.fbXPlanarMover[1].stMoverRef.MCTOPLC/SETONTRACK <-> McToPlc/SETONTRACK
//     PlcTask Inputs/MAIN.fbXMotionUnit.fbXPlanarMover[1].stMoverRef.MCTOPLC/STD <-> McToPlc/STD
//     PlcTask Outputs/MAIN.fbXMotionUnit.fbXPlanarMover[1].stMoverRef.PLCTOMC/STD <-> PlcToMc/STD
//   DMMS_PLC/DMMS_PLC Instance <-> XPlanar MC Project/Axes/0000lcle
//     PlcTask Inputs/MAIN.fbXMotionUnit.fbXPlanarMover[2].stMoverRef.MCTOPLC/ACT <-> McToPlc/ACT
//     PlcTask Inputs/MAIN.fbXMotionUnit.fbXPlanarMover[2].stMoverRef.MCTOPLC/COORDMODE <-> McToPlc/COORDMODE
//     PlcTask Inputs/MAIN.fbXMotionUnit.fbXPlanarMover[2].stMoverRef.MCTOPLC/SET <-> McToPlc/SET
//     PlcTask Inputs/MAIN.fbXMotionUnit.fbXPlanarMover[2].stMoverRef.MCTOPLC/SETONTRACK <-> McToPlc/SETONTRACK
//     PlcTask Inputs/MAIN.fbXMotionUnit.fbXPlanarMover[2].stMoverRef.MCTOPLC/STD <-> McToPlc/STD
//     PlcTask Outputs/MAIN.fbXMotionUnit.fbXPlanarMover[2].stMoverRef.PLCTOMC/STD <-> PlcToMc/STD
//   DMMS_PLC/DMMS_PLC Instance <-> XPlanar MC Project/Groups/CloseLoopTrack
//     PlcTask Inputs/MAIN.fbXMotionUnit.fbCloseLoopTrack.fbTrackStandard.stTrackRef.MCTOPLC_STD <-> McToPlc/STD
//   DMMS_PLC/DMMS_PLC Instance <-> XPlanar MC Project/Groups/Environment
//     PlcTask Inputs/MAIN.fbXMotionUnit.fbXPlanarSystem.environment.MCTOPLC_STD <-> McToPlc/STD
//   DMMS_PLC/DMMS_PLC Instance <-> XPlanar MC Project/Groups/PipetteBufferConTrack
//     PlcTask Inputs/MAIN.fbXMotionUnit.fbTrackPipetteBufferCon.fbTrackStandard.stTrackRef.MCTOPLC_STD <-> McToPlc/STD
//   DMMS_PLC/DMMS_PLC Instance <-> XPlanar MC Project/Groups/PipettePostBufferTrack
//     PlcTask Inputs/MAIN.fbXMotionUnit.fbTrackPipettePostBuffer.fbTrackStandard.stTrackRef.MCTOPLC_STD <-> McToPlc/STD
//   DMMS_PLC/DMMS_PLC Instance <-> XPlanar MC Project/Groups/PipettePreBufferTrack
//     PlcTask Inputs/MAIN.fbXMotionUnit.fbTrackPipettePreBuffer.fbTrackStandard.stTrackRef.MCTOPLC_STD <-> McToPlc/STD
//   DMMS_PLC/DMMS_PLC Instance <-> XPlanar MC Project/Groups/PipetteTrack
//     PlcTask Inputs/MAIN.fbXMotionUnit.fbTrackPipette.fbTrackStandard.stTrackRef.MCTOPLC_STD <-> McToPlc/STD
//   DMMS_PLC/DMMS_PLC Instance <-> XPlanar MC Project/Groups/PuncherBufferTrack
//     PlcTask Inputs/MAIN.fbXMotionUnit.fbTrackBufferPuncher.fbTrackStandard.stTrackRef.MCTOPLC_STD <-> McToPlc/STD
//   DMMS_PLC/DMMS_PLC Instance <-> XPlanar MC Project/Groups/PuncherSeperateTrack
//     PlcTask Inputs/MAIN.fbXMotionUnit.fbPuncherSeperate.fbTrackStandard.stTrackRef.MCTOPLC_STD <-> McToPlc/STD
//   DMMS_PLC/DMMS_PLC Instance <-> XPlanar MC Project/Groups/PuncherWellplateTrack
//     PlcTask Inputs/MAIN.fbXMotionUnit.fbTrackPuncherWellplate.fbTrackStandard.stTrackRef.MCTOPLC_STD <-> McToPlc/STD
//   DMMS_PLC/DMMS_PLC Instance <-> XPlanar MC Project/Groups/StradeFirstSegTrack
//     PlcTask Inputs/MAIN.fbXMotionUnit.fbTrackStradeFirstSeg.fbTrackStandard.stTrackRef.MCTOPLC_STD <-> McToPlc/STD
//   DMMS_PLC/DMMS_PLC Instance <-> XPlanar MC Project/Groups/StradeSecondSegTrack
//     PlcTask Inputs/MAIN.fbXMotionUnit.fbTrackStradeSecondSeg.fbTrackStandard.stTrackRef.MCTOPLC_STD <-> McToPlc/STD
//   DMMS_PLC/DMMS_PLC Instance <-> XPlanar MC Project/Groups/UserInteractionTrack
//     PlcTask Inputs/MAIN.fbXMotionUnit.fbTrackUserInteraction.fbTrackStandard.stTrackRef.MCTOPLC_STD <-> McToPlc/STD
//   DMMS_PLC/DMMS_PLC Instance <-> XPlanar MC Project/Groups/XPlanar
//     PlcTask Inputs/MAIN.fbXMotionUnit.fbXPlanarSystem.group.MCTOPLC_STD <-> McToPlc/STD

// ---- DUTs/Communiction/Movers/ST_ComIn_ExportMover.TcDUT
{attribute 'pack_mode' := '1'}  // needed for python pyads reading
TYPE ST_ComIn_ExportMover :
STRUCT
	Enable:BOOL;
	Reset:BOOL;	
	MoverType:INT;
	ControlWord: INT; 
	TaskToProcessed: UDINT;
	id: STRING(13); 
	WellplateData: ST_WellplateParametrization;
	
	
	
	
END_STRUCT
END_TYPE

// ---- DUTs/Communiction/Movers/ST_ComOut_ExportMover.TcDUT
{attribute 'pack_mode' := '1'}  // needed for python pyads reading
TYPE ST_ComOut_ExportMover :
STRUCT
	Avaiable: BOOL; 
	Error: BOOL;
	CurrentTaskFinished:BOOL;
	Status_Word: INT; 
	Error_ID: INT;
	MoverType:INT;
	CurrentStation: UINT;
	LastTask: UDINT; 
	CurrentTask: UDINT; 
	TrackID: UDINT;
	TrackPos: LREAL;
	Id: STRING(13);
	Position : MoverPositionUnion;
	PartTracking: ST_PartTrackingData;


END_STRUCT
END_TYPE

// ---- DUTs/Communiction/Movers/ST_PartTrackingData.TcDUT
{attribute 'pack_mode' := '1'}  // needed for python pyads reading
TYPE ST_PartTrackingData :
STRUCT
	OK_ToProcess: BOOL;
	NOK_ToProcess: BOOL;
	bInitRun: BOOL;
	WellplateStatus: INT;
	WellplateNOK_Reason: INT;
	nDestinationProcess: UINT;
	nPriority: UINT;
	nSerial: UDINT;
	PuncherProcessResults: ARRAY[1..96] OF ST_ProcessResult;
	PipeteProcesResults: ARRAY[1..96] OF ST_ProcessResult;
	DoseProcesResult: ARRAY[1..12] OF ST_ProcessResult;
END_STRUCT
END_TYPE

// ---- DUTs/Communiction/Movers/ST_Com_ExportMover.TcDUT
{attribute 'pack_mode' := '1'}  // needed for python pyads reading
TYPE ST_Com_ExportMover :
STRUCT
		IN: 			ST_ComIn_ExportMover;
		OUT:			ST_ComOut_ExportMover;
		ProcessData:	ST_ProductData;
		ManualMovements:ST_ManualMovements;
END_STRUCT
END_TYPE

// ---- DUTs/Communiction/Station/ST_ComIn_ExportStation.TcDUT
{attribute 'pack_mode' := '1'}  // needed for python pyads reading
TYPE ST_ComIn_ExportStation :
STRUCT
	Enable: BOOL;
	StationName: INT;
	ControlWord: INT;
END_STRUCT
END_TYPE

// ---- DUTs/Communiction/Station/ST_ComOut_ExportStation.TcDUT
{attribute 'pack_mode' := '1'}  // needed for python pyads reading
TYPE ST_ComOut_ExportStation :
STRUCT
	Enable: BOOL;
	ProcessComplete: BOOL;
	OK: BOOL;
	NOK: BOOL;
	Error: BOOL;
	StatusWord: INT;
	StationName: INT;
	Error_ID: INT;
	ProcesedMover: STRING(13);
	MoversList: ARRAY[1..10] OF STRING(13);
END_STRUCT
END_TYPE

// ---- DUTs/Communiction/Station/ST_EStationName.TcDUT
{attribute 'qualified_only'}
{attribute 'strict'}
{attribute 'to_string'}
TYPE ST_EStationName :
(
	ST01 := 1,
	ST02 := 2,
	ST03 := 3,
	ST04 := 4,
	ST05 := 5,
	ST06 := 6
);
END_TYPE

// ---- DUTs/Communiction/Station/ST_ManMov_Station.TcDUT
{attribute 'pack_mode' := '1'}  // needed for python pyads reading
TYPE ST_ManMov_Station :
STRUCT
	CMD: INT;
	CMD_Confirm: INT;
	CMD_done: BOOL;
END_STRUCT
END_TYPE

// ---- DUTs/Communiction/Station/ST_Com_ExportStation.TcDUT
TYPE ST_Com_ExportStation :
STRUCT
		IN: 		ST_ComIn_ExportStation;
		OUT:		ST_ComOut_ExportStation;
		ManualMovement: ST_ManMov_Station;
END_STRUCT
END_TYPE

// ---- Mover/DUTs/ST_ControlData.TcDUT
{attribute 'pack_mode' := '1'}
TYPE ST_ControlData :
STRUCT
	StatusWord: INT;
	ControlWord: INT;
END_STRUCT
END_TYPE

// ---- Mover/DUTs/ST_EMoverLoadType.TcDUT
{attribute 'qualified_only'}
{attribute 'strict'}
{attribute 'to_string'}
TYPE ST_EMoverLoadType :
(
	Wellplate := 1,
	PipetteTips:=2,
	Gripper:=3
);
END_TYPE

// ---- Mover/DUTs/ST_ManMov_MoveTrack.TcDUT
{attribute 'pack_mode' := '1'}  // needed for python pyads reading
TYPE ST_ManMov_MoveTrack :
STRUCT
	move_track_CMD_enable:BOOL;
	move_track_CMD_done:BOOL;
	// Commands
	join_track:BOOL;
	leave_track:BOOL;
	move_track:BOOL; 
	
	//moving settings
	move_track_no: INT;	
	move_track_position: REAL; 

END_STRUCT
END_TYPE

// ---- Mover/DUTs/ST_ProcessTask.TcDUT
{attribute 'pack_mode' := '1'}  // needed for python pyads reading
TYPE ST_ProcessTask :
STRUCT
	CurrentTaskFinished: BOOL;
	LastTask: UDINT;
	TaskToProcessed: UDINT;
	CurrentTask: UDINT;

END_STRUCT
END_TYPE

// ---- Mover/DUTs/ST_ProductData.TcDUT
{attribute 'pack_mode' := '1'}  // needed for python pyads reading
TYPE ST_ProductData :
STRUCT
	
	OK_ToProcess		:BOOL;
	NOK_ToProcess		:BOOL; 
	bInitRun			:BOOL;
	WellplateStatus		:INT;
	WellplateNOK_Reason	:INT;
	nDestinationProcess	:UINT;
	nPriority			:UINT;
	nSerial				:UDINT;
	PuncherProcessResults 	: ARRAY[1..96] OF ST_ProcessResult;
	PipeteProcesResults		: ARRAY [1..96] OF ST_ProcessResult;
	

END_STRUCT
END_TYPE

// ---- Mover/DUTs/ST_WellplateParametrization.TcDUT
{attribute 'pack_mode' := '1'}  // needed for python pyads reading
TYPE ST_WellplateParametrization :
STRUCT
	Row: INT;
	Columns:INT;
	DistanceBetweenHoles_X:REAL;
	DistanceBetweenHoles_Y:REAL;
	OffsetFirstHoles_X:REAL; 
	OffsetFirstHoles_Y:REAL; 
 
	
END_STRUCT
END_TYPE

// ---- Stations/DUTs/ST_EStationProcessState.TcDUT
{attribute 'qualified_only'}
{attribute 'strict'}
{attribute 'to_string'}
TYPE ST_EStationProcessState :
(	
	Empty := 1,
	InProcess:=2,
	Finished:=3
);
END_TYPE

// ---- Stations/DUTs/ST_StationPosition.TcDUT
TYPE ST_StationPosition :
STRUCT
	bInit				: BOOL;
	fPositionOnTrack	: LREAL;
	nTrackId			: UINT;
	fPosition_X			: LREAL;
	fPosition_Y			: LREAL;
END_STRUCT
END_TYPE

// ---- Stations/DUTs/ST_VisStationData.TcDUT
TYPE ST_VisStationData :

STRUCT
	
	bInit		: BOOL;
	fPosition_X	: LREAL;
	fPosition_Y : LREAL;

END_STRUCT

END_TYPE

// ---- GVLs/Communication.TcGVL
{attribute 'qualified_only'}
VAR_GLOBAL
	RunAplicationComm: bool; 

	StopApplicationComm: BOOL;

	g_Com_GlobalState: ST_Com_GlobalStatus;

	g_Com_Movers : ARRAY[1..GVL.gc_nMaxNumberMovers] OF ST_Com_ExportMover;
	
	g_Com_Stations : ARRAY[1..GVL.gc_NumberStations] OF ST_Com_ExportStation;



	std: INT;
	Init: INT;
END_VAR

// ---- GVLs/GVL.TcGVL
{attribute 'qualified_only'}
VAR_GLOBAL CONSTANT
	
	gc_nMaxNumberMovers			: UDINT := 2;	
	gc_nMoverCountConfigured 	: UDINT := gc_nMaxNumberMovers;
	
	gc_MaxNumberTiles			: UDINT := 5;

	gc_NumberTracks				: UDINT := 11;		// Number of tracks controlled by the application
	gc_NumberStations			: UINT  := 3;		// Number of stations controlled by the application


// track numeration

		TrackPuncherWellplate	: UDINT := 1;
		TrackStradeFirstSeg		: UDINT := 2;
		TrackStradeSecondSeg	: UDINT := 3;
		TrackBufferPuncher		: UDINT := 4;
		TrackPipettePreBuffer   : UDINT := 5;
		TrackPipette			: UDINT := 6;
		TrackPipettePostBuffer	: UDINT := 7;
		TrackPipetteBufferCon	: UDINT := 8;
		TrackUserInteraction	: UDINT := 9;
		CloseLoopTrack			: UDINT := 10;
		PuncherSeperateTrack	: UDINT	:= 11;
		

// station numeration 
		PuncherStation			: UDINT := 1;
		PuncherSeparateStation	: UDINT := 2;
		PuncherBufferStation	: UDINT := 3;
		
// mover calibration 
		stPayloadWellplateDown	: 	ST_TcIoPayload:=(
									AAxisInertia:=0.00096045220,
									BAxisInertia:=0.00110988871,
									CAxisInertia :=0.00140891283,
									CentreOfMassX :=0,
									CentreOfMassY:= 0,
									CentreOfMassZ:=25.74,
									Mass:=0.45194 );
		
		stPayloadWellplateMiddle: 	ST_TcIoPayload:=(
									AAxisInertia:=0.00098632707,
									BAxisInertia:= 0.00113576347,
									CAxisInertia :=0.00140891283,
									CentreOfMassX :=0,
									CentreOfMassY:= 0,
									CentreOfMassZ:=33.23,
									Mass:=0.45194 );
									
		stPayloadWellplateUp	: 	ST_TcIoPayload:=(
									AAxisInertia:= 0.00117197,
									BAxisInertia:=0.00132141,
									CAxisInertia :=0.00140891,
									CentreOfMassX :=0,
									CentreOfMassY:= 0,
									CentreOfMassZ:=0,
									Mass:=0 );
		
		stPayloadGripper		: 	ST_TcIoPayload:=(
									AAxisInertia:=0,
									BAxisInertia:=0,
									CAxisInertia :=0,
									CentreOfMassX :=0,
									CentreOfMassY:= 0,
									CentreOfMassZ:=0,
									Mass:=0 );
		
		stPayloadPipetteTips	: 	ST_TcIoPayload:=(
									AAxisInertia:=0,
									BAxisInertia:=0,
									CAxisInertia :=0,
									CentreOfMassX :=0,
									CentreOfMassY:= 0,
									CentreOfMassZ:=0,
									Mass:=0 );



END_VAR

VAR_GLOBAL
	g_nMoverCount : UDINT ;
	g_Tracks : ARRAY[1..gc_NumberTracks] OF I_Track;
	g_Stations : ARRAY[1..gc_NumberStations] OF I_Station;
	g_Movers : ARRAY[1..gc_nMaxNumberMovers] OF I_MoverApplication;
	
END_VAR

// ---- Mover/I_MoverApplication.TcIO
INTERFACE I_MoverApplication

METHOD Cycle
END_METHOD

METHOD ManualMovement : BOOL
VAR_INPUT
	bReset: bool;
END_VAR
END_METHOD

PROPERTY P_ControlData : Reference to ST_ControlData
GET
END_GET
SET
END_SET
END_PROPERTY

PROPERTY P_MoverConfiguration : Reference to  ST_MoverConfiguration
GET
END_GET
SET
END_SET
END_PROPERTY

PROPERTY P_MoverID : STRING
GET
END_GET
SET
END_SET
END_PROPERTY

PROPERTY P_MoverIndex : INT
GET
END_GET
SET
END_SET
END_PROPERTY

PROPERTY P_ProcessTask :  ST_ProcessTask
GET
END_GET
SET
END_SET
END_PROPERTY

PROPERTY P_ProductData : Reference to ST_ProductData
GET
END_GET
SET
END_SET
END_PROPERTY

PROPERTY P_TrackId : UDINT
GET
END_GET
SET
END_SET
END_PROPERTY

PROPERTY P_CurrentStation : UINT
GET
END_GET
SET
END_SET
END_PROPERTY

PROPERTY P_Enable : BOOL
GET
END_GET
SET
END_SET
END_PROPERTY

PROPERTY P_Error : BOOL
GET
END_GET
SET
END_SET
END_PROPERTY

PROPERTY P_ErrorID : INT
GET
END_GET
SET
END_SET
END_PROPERTY

PROPERTY P_TrackPos : LREAL
GET
END_GET
SET
END_SET
END_PROPERTY

PROPERTY P_PartTracking : ST_PartTrackingData
GET
END_GET
SET
END_SET
END_PROPERTY

PROPERTY std : I_XPlanarMoverStandard
GET
END_GET
SET
END_SET
END_PROPERTY

END_INTERFACE

// ---- Stations/Base/I_Station.TcIO
INTERFACE I_Station

METHOD Clear : BOOL
VAR_INPUT
END_VAR
END_METHOD

METHOD Cycle : BOOL
VAR_INPUT
END_VAR
END_METHOD

METHOD Init : BOOL
END_METHOD

PROPERTY P_bInitDone : BOOL
GET
END_GET
END_PROPERTY

PROPERTY P_eProcessMode : E_ProcessMode
GET
END_GET
SET
END_SET
END_PROPERTY

PROPERTY P_List_Station : I_List
GET
END_GET
END_PROPERTY

PROPERTY P_List_Switch_Input_E : I_List
GET
END_GET
END_PROPERTY

PROPERTY P_List_Switch_Input_N : I_List
GET
END_GET
END_PROPERTY

PROPERTY P_List_Switch_Input_S : I_List
GET
END_GET
END_PROPERTY

PROPERTY P_List_Switch_Input_W : I_List
GET
END_GET
END_PROPERTY

PROPERTY P_nErrorCode : UDINT
GET
END_GET
END_PROPERTY

PROPERTY P_Position : ST_StationPosition
GET
END_GET
END_PROPERTY

PROPERTY P_ProcessClearance : DINT
GET
END_GET
END_PROPERTY

PROPERTY P_ProcessRequest : UDINT
GET
END_GET
SET
END_SET
END_PROPERTY

PROPERTY P_ProcessState : UDINT
GET
END_GET
END_PROPERTY

PROPERTY P_StationTaskList : array[1..200] of UDINT
GET
END_GET
SET
END_SET
END_PROPERTY

METHOD Process : BOOL
END_METHOD

END_INTERFACE

// ---- Mover/FB_ApplicationMover.TcPOU
FUNCTION_BLOCK FB_ApplicationMover IMPLEMENTS I_MoverApplication
VAR
	ipMoverStandard	: I_XPlanarMoverStandard;
	
	stProductData	: ST_ProductData;
	eMoverType 		: ST_EMoverLoadType;
	
	nMoverIndex		: INT;
	sMoverID 		: STRING(13) := '00001111';
	
	nTrackId		: UDINT;
	
	// customer Data
	bIsLoaded		: BOOL;	
	stControlData	:ST_ControlData;
	stMoverConfiguration: ST_MoverConfiguration;
	stProcessTask: St_ProcessTask;
	nCurrentStation	: UINT;
	bEnable			: BOOL;
	bError			: BOOL;
	nErrorID		: INT;
	stPartTracking	: ST_PartTrackingData;
	rTrackPos		: LREAL;



END_VAR

METHOD Cycle


VAR_INST
	nTestCounter	: UINT;
	index: UDINT;
	
END_VAR
IF std <> 0 THEN

    std.cycle();

    IF communication.RunAplicationComm THEN 
        FOR index := 1 TO GVL.gc_nMaxNumberMovers DO 

            IF communication.g_Com_Movers[index].IN.id = THIS^.P_MoverID THEN 

                //================= OUT =================

                Communication.g_Com_Movers[index].OUT.Avaiable := (THIS^.std.P_State = 3); // Avaiable

                Communication.g_Com_Movers[index].OUT.Error := THIS^.P_Error; // Error

                Communication.g_Com_Movers[index].OUT.CurrentTaskFinished := stProcessTask.CurrentTaskFinished; // CurrentTaskFinished

                stControlData.StatusWord := THIS^.std.P_State;
                Communication.g_Com_Movers[index].OUT.Status_Word := stControlData.StatusWord; // Status_Word

                Communication.g_Com_Movers[index].OUT.Error_ID := THIS^.P_ErrorID; // Error_ID

                communication.g_Com_Movers[index].out.MoverType := THIS^.stMoverConfiguration.MoverType; // MoverType

                Communication.g_Com_Movers[index].OUT.CurrentStation := THIS^.P_CurrentStation; // CurrentStation

                Communication.g_Com_Movers[index].OUT.LastTask := stProcessTask.LastTask; // LastTask
                Communication.g_Com_Movers[index].OUT.CurrentTask := stProcessTask.CurrentTask; // CurrentTask

                Communication.g_Com_Movers[index].OUT.TrackID := THIS^.P_TrackId; // TrackID

                Communication.g_Com_Movers[index].OUT.TrackPos := THIS^.P_TrackPos; // TrackPos

                Communication.g_Com_Movers[index].OUT.Id := THIS^.P_MoverID; // Id

                Communication.g_Com_Movers[index].OUT.position.vec := THIS^.std.P_ActPosition;
                Communication.g_Com_Movers[index].OUT.Position.vec.x := THIS^.std.P_ActPosition.x;
                Communication.g_Com_Movers[index].OUT.Position.vec.y := THIS^.std.P_ActPosition.y;
                Communication.g_Com_Movers[index].OUT.Position.vec.c := THIS^.std.P_ActPosition.c; // Position

                Communication.g_Com_Movers[index].OUT.PartTracking := THIS^.P_PartTracking; // Part tracking

                //================= IN =================

                THIS^.P_Enable := Communication.g_Com_Movers[index].IN.Enable; // Enable

                IF Communication.g_Com_Movers[index].IN.Reset THEN
                    ipMoverStandard.Reset(slogMessage := 'mover reset');
                END_IF // Reset

                stMoverConfiguration.MoverType := Communication.g_Com_Movers[index].IN.MoverType;
                IF communication.g_Com_Movers[index].IN.MoverType = 1 THEN 
                    eMoverType := ST_EMoverLoadType.Wellplate;
                ELSIF communication.g_Com_Movers[index].IN.MoverType = 2 THEN 
                    eMoverType := ST_EMoverLoadType.Gripper;
                ELSIF communication.g_Com_Movers[index].IN.MoverType = 3 THEN 
                    eMoverType := ST_EMoverLoadType.PipetteTips;
                END_IF	// Mover Type

                stControlData.ControlWord := communication.g_Com_Movers[index].IN.ControlWord; // ControlWord

                stProcessTask.TaskToProcessed := Communication.g_Com_Movers[index].IN.TaskToProcessed; // TaskToProcced

                // ID — użyte wyżej do dopasowania slotu

                stMoverConfiguration.WellplateData := Communication.g_Com_Movers[index].IN.WellplateData; // WellplateData

            END_IF
        END_FOR
    END_IF

END_IF
END_METHOD

METHOD ManualMovement : BOOL
VAR_INPUT
	bReset: bool;
END_VAR

VAR_INST
	nTestCounter	: UINT;
	index: UDINT;
	Com_Index: UDINT;
	nMovementSequence : UDINT;
	
	
END_VAR

VAR
	ManMovements: 	ST_ManualMovements;
	targetPos 						:  PositionXYC;
	fTargetPosOnTrack 				: LREAL;
	stOptionsJoinTrack				: ST_JoinTrackOptions;
	stMoveOnTrackOptions			: ST_MoveOnTrackOptions;
	stMoveToPositionOptions			: ST_MoveToPositionOptions;
	bMoversJoined 					: BOOL;
	bMoverError						: BOOL;
	bMoversInPos					: BOOL;
	strInfo							: STRING;
	
END_VAR
	IF communication.RunAplicationComm THEN 
		FOR index:=1 TO GVL.gc_nMaxNumberMovers DO 
			
			IF communication.g_Com_Movers[index].IN.id= THIS^.P_MoverID THEN
				
				ManMovements:= communication.g_Com_Movers[index].ManualMovements;
				Com_Index:=index;
				
			END_IF
			
		END_FOR
		
	END_IF
	
	
	
	IF bReset OR  Communication.g_Com_GlobalState.IN.Stop   OR Communication.g_Com_GlobalState.IN.Reset THEN 
	ManualMovement := FALSE;
	nMovementSequence := 0;
END_IF

CASE nMovementSequence OF
	

0: //init
		
 	// wait for enabling  process 
			 IF Communication.g_Com_GlobalState.IN.Start AND NOT Communication.g_Com_GlobalState.IN.EOC_Stop  AND Com_Index <>0 THEN 
				IF Communication.g_Com_GlobalState.IN.ProgramType =2 THEN 
					  nMovementSequence := 100;
				
					   ELSIF Communication.g_Com_GlobalState.IN.ProgramType =3 THEN 
					  nMovementSequence := 200;
				END_IF								
					 
			 END_IF
			 




100:	 // position test 
	
		// leave track
		IF ipMoverStandard.P_CommandMode= MC_PLANAR_MOVER_COMMAND_MODE.OnTrack AND  NOT ipMoverStandard.P_Busy THEN

			ipMoverStandard.LeaveTrackInPosition( strInfo, FALSE);
			nMovementSequence := nMovementSequence +1;
		ELSE 
			nMovementSequence := 110;
		END_IF


101:
			IF ipMoverStandard.P_LeaveTrackInPosition.Done THEN
				P_TrackId:=0;
				nMovementSequence := 110;
			ELSIF ipMoverStandard.P_LeaveTrackInPosition.Error THEN
				nMovementSequence := nMovementSequence +4;
			END_IF	
				


110://setup state 
		IF NOT ManMovements.FreeMove.move_position_CMD_enable THEN 
				ManMovements.FreeMove.move_position_CMD_done:= FALSE;
				communication.g_Com_Movers[Com_Index].ManualMovements:=ManMovements;
		END_IF
						nMovementSequence := nMovementSequence +  1;					  
				
111: 	//execute command 
stMoveToPositionOptions.useOrientation:= TRUE;
	targetPos.x:=	ManMovements.FreeMove.move_position.x ;
	targetPos.y:=	ManMovements.FreeMove.move_position.y;
	targetPos.C:=	ManMovements.FreeMove.move_position.C;
					 // targetpos.ShiftByXy(ManMovements.move_position.x,ManMovements.move_position.y);
				
	


			IF  ManMovements.FreeMove.move_position_CMD_enable AND NOT ManMovements.FreeMove.move_position_CMD_done  THEN 
					ipMoverStandard.MoveToPositionEXt('move to XY', targetPos, 100, 2500, 2500, 25000,stMoveToPositionOptions);
					nMovementSequence := nMovementSequence +  1;
			ELSE
				nMovementSequence := 0;
			END_IF
				
		
	
	
112: 	// check commad result 

		
		IF ipMoverStandard.P_MoveToPositionExt.Done THEN
			ManMovements.FreeMove.move_position_CMD_done:= TRUE;
			communication.g_Com_Movers[Com_Index].ManualMovements:=ManMovements;
			nMovementSequence :=  0;
		ELSIF ipMoverStandard.P_MoveToPositionExt.Error THEN
			nMovementSequence := nMovementSequence +  3;
		END_IF				
		
		
200:
		 IF NOT ManMovements.MoveTrack.move_track_CMD_done THEN 
				IF ManMovements.MoveTrack.join_track AND ManMovements.MoveTrack.move_track_no<>0 THEN 
					nMovementSequence := 210;
				ELSIF ManMovements.MoveTrack.leave_track THEN
					nMovementSequence := 220;
				ELSIF ManMovements.MoveTrack.move_track AND ManMovements.MoveTrack.move_track_no<>0 THEN 
					nMovementSequence := 230;
				ELSE
					nMovementSequence := 0;
				END_IF
		END_IF
		
		IF NOT ManMovements.MoveTrack.move_track_CMD_enable THEN 
			ManMovements.MoveTrack.move_track_CMD_done := FALSE;
			communication.g_Com_Movers[Com_Index].ManualMovements:=ManMovements;
		END_IF

210:	
		stOptionsJoinTrack.useOrientation := TRUE;
	
		IF (ipMoverStandard.P_CommandMode<> MC_PLANAR_MOVER_COMMAND_MODE.OnTrack OR  INT_TO_UDINT(ManMovements.MoveTrack.move_track_no)<>P_TrackId)
			AND NOT ipMoverStandard.P_Busy
			AND ManMovements.MoveTrack.move_track_CMD_enable THEN
			ipMoverStandard.JoinTrack('Joining track', GVL.g_Tracks[ManMovements.MoveTrack.move_track_no].std, 250, 1250, 12500, stOptionsJoinTrack);
				nMovementSequence := nMovementSequence + 1;
			ELSE 
				nMovementSequence := 0;
		END_IF
	
	
		
211:
	
			bMoversJoined := ipMoverStandard.P_JoinTrack.Done;
			bMoverError :=  ipMoverStandard.P_JoinTrack.Error;			
		
	IF bMoversJoined THEN
		ManMovements.MoveTrack.move_track_CMD_done:=TRUE;
		communication.g_Com_Movers[Com_Index].ManualMovements:=ManMovements;
		P_TrackId:=INT_TO_UDINT(ManMovements.MoveTrack.move_track_no);
		nMovementSequence := 0;
	ELSIF bMoverError THEN
 			nMovementSequence := nMovementSequence + 4;
	END_IF

		
	
		
220:
		
		IF ipMoverStandard.P_CommandMode= MC_PLANAR_MOVER_COMMAND_MODE.OnTrack AND  NOT ipMoverStandard.P_Busy AND ManMovements.MoveTrack.move_track_CMD_enable  THEN

			ipMoverStandard.LeaveTrackInPosition( strInfo, FALSE);
			nMovementSequence := nMovementSequence +1;
		ELSE 
			nMovementSequence := 0;
		END_IF


221:
			IF ipMoverStandard.P_LeaveTrackInPosition.Done THEN
				ManMovements.MoveTrack.move_track_CMD_done:=TRUE;
				communication.g_Com_Movers[Com_Index].ManualMovements:=ManMovements;
				P_TrackId:=0;
				nMovementSequence := 0;
			ELSIF ipMoverStandard.P_LeaveTrackInPosition.Error THEN
				nMovementSequence := nMovementSequence +4;
			END_IF	
			
230:

		
		stMoveOnTrackOptions.gap := 120;
		fTargetPosOnTrack:=ManMovements.MoveTrack.move_track_position;
		stMoveOnTrackOptions.dynamicMode := MC_DYNAMICS_REDUCTION_MODE.AccelerationLimitedVelocity;
		stMoveOnTrackOptions.direction := MC_DIRECTION.mcDirectionShortestWay;
		IF   NOT ipMoverStandard.P_Busy AND ManMovements.MoveTrack.move_track_CMD_enable  THEN
				 ipMoverStandard.MoveOnTrackEXT('move on track', GVL.g_Tracks[ManMovements.MoveTrack.move_track_no].std, fTargetPosOnTrack,
								300, 3000, 15000, stMoveOnTrackOptions);
				nMovementSequence := nMovementSequence +1;
		 END_IF
		 


	231:
			bMoversInPos :=  ipMoverStandard.P_MoveOnTrackExt.Done;
			bMoverError := ipMoverStandard.P_MoveOnTrackExt.Error;
	
		
		IF bMoversInPos THEN
			ManMovements.MoveTrack.move_track_CMD_done:=TRUE;
			communication.g_Com_Movers[Com_Index].ManualMovements:=ManMovements;
			nMovementSequence := 0;
		ELSIF bMoverError THEN
			nMovementSequence := nMovementSequence +  3;
		END_IF
			
			
			
	END_CASE
END_METHOD

PROPERTY P_ControlData : Reference to ST_ControlData
GET
P_ControlData := stControlData;
END_GET
SET
stControlData := P_ControlData;
END_SET
END_PROPERTY

PROPERTY P_CurrentStation : UINT
GET
P_CurrentStation := nCurrentStation;
END_GET
SET
nCurrentStation := P_CurrentStation;
END_SET
END_PROPERTY

PROPERTY P_Enable : BOOL
GET
P_Enable := bEnable;
END_GET
SET
bEnable := P_Enable;
END_SET
END_PROPERTY

PROPERTY P_Error : BOOL
GET
P_Error := bError;
END_GET
SET
bError := P_Error;
END_SET
END_PROPERTY

PROPERTY P_ErrorID : INT
GET
P_ErrorID := nErrorID;
END_GET
SET
nErrorID := P_ErrorID;
END_SET
END_PROPERTY

PROPERTY P_MoverConfiguration : Reference to  ST_MoverConfiguration
GET
P_MoverConfiguration := stMoverConfiguration;
END_GET
SET
stMoverConfiguration := P_MoverConfiguration;
END_SET
END_PROPERTY

PROPERTY P_MoverID : STRING
GET
P_MoverID := sMoverID;
END_GET
SET
sMoverID := P_MoverID;
END_SET
END_PROPERTY

PROPERTY P_MoverIndex : INT
GET
P_MoverIndex := nMoverIndex;
END_GET
SET
nMoverIndex := P_MoverIndex;
END_SET
END_PROPERTY

PROPERTY P_PartTracking : ST_PartTrackingData
GET
P_PartTracking := stPartTracking;
END_GET
SET
stPartTracking := P_PartTracking;
END_SET
END_PROPERTY

PROPERTY P_ProcessTask : ST_ProcessTask
GET
P_ProcessTask := stProcessTask;
END_GET
SET
stProcessTask := P_ProcessTask;
END_SET
END_PROPERTY

PROPERTY P_ProductData : Reference to ST_ProductData
GET
P_ProductData REF= stProductData;
END_GET
SET
stProductData := P_ProductData;
END_SET
END_PROPERTY

PROPERTY P_TrackId : UDINT
GET
P_TrackId := nTrackId;
END_GET
SET
nTrackId := P_TrackId;
END_SET
END_PROPERTY

PROPERTY P_TrackPos : LREAL
GET
P_TrackPos := rTrackPos;
END_GET
SET
rTrackPos := P_TrackPos;
END_SET
END_PROPERTY

PROPERTY std : I_XPlanarMoverStandard
GET
IF ipMoverStandard <> 0 THEN
	std := ipMoverStandard;	
END_IF
END_GET
SET
ipMoverStandard := std;
END_SET
END_PROPERTY

END_FUNCTION_BLOCK

// ---- POUs/FB_MotionSystem.TcPOU
FUNCTION_BLOCK FB_MotionSystem
VAR_INPUT
END_VAR
VAR_OUTPUT
END_VAR
VAR
	fbXPlanarSystem	: FB_XPlanarSystem;
	stMoverDetectionInfos   : ST_TcIoMoverDetectionInfos;
	fbTcIoXPlanarEnv	:FB_TcIoXPlanarEnvironment  ; 
	ipXpu	: I_TcIoXPlanarProcessingUnit;

	
	fbMover					: ARRAY [1..GVL.gc_nMaxNumberMovers] OF FB_ApplicationMover;
	fbXPlanarMover : ARRAY [1..GVL.gc_nMaxNumberMovers] OF FB_XPlanarMoverStandard; 
	
	nStartupSequence : UDINT;
	nStartingSequence : UDINT;
	nExecutingSequence : UDINT;
	nResettingSequence 	: UDINT;
	nRecoverySequence : UDINT;
	
	// Helper
	bDone 					: BOOL;
	idx						: UDINT;
	nForCounter 			: UDINT;	
	nErrorID				: UDINT;
	bMoverError				: BOOL;	
	
	// TRACKS
	fbTrackPuncherWellplate		: FB_PuncherWellplateTrack;
	fbTrackBufferPuncher		: FB_PuncherBufferTrack;
	fbPuncherSeperate			: FB_PuncherSeperateTrack;
	fbTrackStradeFirstSeg		: FB_StradeFirstSegTrack;
	fbTrackStradeSecondSeg		: FB_StradeSecondSegTrack;
	fbTrackPipettePreBuffer		: FB_PipettePreBufferTrack;
	fbTrackPipette				: FB_PipetteTrack;
	fbTrackPipettePostBuffer	: FB_PipettePostBufferTrack;
	fbTrackPipetteBufferCon		: FB_PipetteBufferConTrack;
	fbTrackUserInteraction		: FB_UserInteractionTrack;
	fbCloseLoopTrack			: FB_CloseLoopTrack;

	
	// STATIONS
	fbPuncherStation : FB_PuncherStation;
	fbPuncherSeparateStation : FB_PuncherSeparateStation;
	fbPuncherBufferStation : FB_PuncherBufferStation;
	
	bAssignmentComplete 		: BOOL;
	

	
END_VAR

METHOD Cycle
VAR_INPUT
END_VAR

VAR
	index	: UDINT;
END_VAR

fbXPlanarSystem.Cycle();

IF bAssignmentComplete THEN

	FOR index := 1 TO  MoverCount DO
		fbXPlanarMover[index].Cycle();
		GVL.g_Movers[index].Cycle();
		fbMover[index].Cycle();
	END_FOR

	FOR index := 1 TO GVL.gc_NumberTracks DO
		GVL.g_Tracks[index].Cycle();
	END_FOR
	IF DEBUG.IBN_bool[1] THEN
		FOR index := 1 TO GVL.gc_NumberStations DO
			GVL.g_Stations[index].Cycle();
		END_FOR
	END_IF
END_IF
END_METHOD

METHOD Execute : BOOL
VAR_INPUT
	bReset : BOOL;
END_VAR

VAR
	index : UDINT;
	com_index:UDINT;
	stMoveOnTrackOptions: ST_MoveOnTrackOptions;
END_VAR

VAR_INST
	
	stOptionsJoinTrack				: ST_JoinTrackOptions;
	bMoversJoined 					: BOOL;
	nMoverToTurnBack				: UDINT;
	nTrackToCheck					:UDINT; 
	nDistanceToTrack				:LREAL;
	nDistanceToTargetTrack			: ARRAY[1..moverCount] OF REAL;
	nTargetTrack					: ARRAY[1..moverCount] OF UDINT;
	bMoversinPos					:BOOL;
	bMoverError						:BOOL;
	stMoverConf					:ST_MoverConfiguration;
	
END_VAR
IF bReset OR  Communication.g_Com_GlobalState.IN.EOC_Stop   THEN
	Execute := FALSE;
	nExecutingSequence := 0;
END_IF

CASE nExecutingSequence OF
	

0: //init
		bMoversinPos := FALSE;
		bMoverError := FALSE;
 	// wait for enabling  process 
			 IF Communication.g_Com_GlobalState.IN.Start AND NOT Communication.g_Com_GlobalState.IN.EOC_Stop THEN 
				 IF Communication.g_Com_GlobalState.IN.ProgramType =1 THEN 
				 nExecutingSequence := 10;
			
				 Communication.g_Com_GlobalState.OUT.ProgramType:=1;
				 
				 ELSIF Communication.g_Com_GlobalState.IN.ProgramType =2 THEN 
					  nExecutingSequence := 20;
					   Communication.g_Com_GlobalState.OUT.InCycle:=FALSE; 
						Communication.g_Com_GlobalState.OUT.ProgramType:=2;
				
					   ELSIF Communication.g_Com_GlobalState.IN.ProgramType =3 THEN 
					  nExecutingSequence := 30;
					  	Communication.g_Com_GlobalState.OUT.InCycle:=FALSE; 
						Communication.g_Com_GlobalState.OUT.ProgramType:=3;
						
				END_IF								
					 
			 END_IF
			 

			 
10:			 // auto cycle 
			// check all movers join to track
			
			FOR index := 1 TO gvl. g_nMoverCount DO
			IF fbXPlanarMover[index].P_CommandMode<> MC_PLANAR_MOVER_COMMAND_MODE.OnTrack THEN 
				
					nExecutingSequence := nExecutingSequence + 1;
					index:=nMoverToTurnBack;
				RETURN ;
			END_IF
			END_FOR 
			nExecutingSequence := nExecutingSequence + 5;
	
11: // look for for nearest track 

	
	FOR index := 1 TO  gvl.g_nMoverCount DO
		nDistanceToTargetTrack[index]:= 999999;
		
		FOR nTrackToCheck :=1 TO GVL.gc_NumberTracks DO 
		nDistanceToTrack := fbXPlanarMover[ index].GetDistanceToTrack(GVL.g_Tracks[nTrackToCheck].std);
		
		IF nDistanceToTrack < nDistanceToTargetTrack[index] AND nDistanceToTrack<> -1 THEN 
			nDistanceToTargetTrack[index]:=nDistanceToTrack;
			nTargetTrack[index] :=nTrackToCheck;
		END_IF
		
		END_FOR
	END_FOR
	
	nExecutingSequence := nExecutingSequence + 1;
	
12: // join to track

		stOptionsJoinTrack.useOrientation := TRUE;
		

		
	FOR index := 1 TO gvl.g_nMoverCount DO
// 		
// 		IF fbXPlanarMover[index].P_CommandMode<> MC_PLANAR_MOVER_COMMAND_MODE.OnTrack THEN
// 			IF  GVL.g_Movers[index].P_MoverConfiguration.MoverType= ST_EMoverLoadType.Wellplate THEN 

				fbXPlanarMover[index].JoinTrack('Joining track', GVL.g_Tracks[nTargetTrack[index]].std, 250, 1250, 12500, stOptionsJoinTrack);
			
// 			ELSIF  GVL.g_Movers[index].P_MoverConfiguration.MoverType= ST_EMoverLoadType.Gripper THEN 
// 					
// 				fbXPlanarMover[index].JoinTrack('Joining track', GVL.g_Tracks[11].std, 250, 1250, 12500, stOptionsJoinTrack);
// 			
// 			ELSIF  GVL.g_Movers[index].P_MoverConfiguration.MoverType= ST_EMoverLoadType.PipetteTips THEN 
// 					
// 				fbXPlanarMover[index].JoinTrack('Joining track', GVL.g_Tracks[7].std, 250, 1250, 12500, stOptionsJoinTrack);
// 			
// 			END_IF
// 		END_IF
// 		
		END_FOR
	
			nExecutingSequence := nExecutingSequence + 1;
		
	13:
		bMoversJoined := TRUE;
		bMoverError := FALSE;
	FOR index := 1 TO moverCount DO
			
			bMoversJoined := bMoversJoined AND fbXPlanarMover[index].P_JoinTrack.Done;
			IF  fbXPlanarMover[index].P_JoinTrack.Done THEN 
				gvl.g_Movers[index].P_TrackId:=nTargetTrack[index];
			END_IF
			bMoverError := bMoverError OR fbXPlanarMover[index].P_JoinTrack.Error;	
			 	
		END_FOR
		
	IF bMoversJoined THEN
			nExecutingSequence := 10;
	ELSIF bMoverError THEN
 			nExecutingSequence := nExecutingSequence + 4;
	END_IF
			
14: 	//send mover to station 
	  	  
		FOR index := 1 TO gvl.g_nMoverCount DO
			 IF fbXPlanarMover[index].P_TrackId= GVL.TrackPuncherWellplate 
			AND GVL.g_Movers[index].P_MoverConfiguration.MoverType= ST_EMoverLoadType.Wellplate
			
			  THEN 
				 fbPuncherStation.P_List_Switch_Input_W.AddMover(GVL.g_Movers[index].std);
			 END_IF

			  IF GVL.g_Movers[index].P_MoverConfiguration.MoverType= ST_EMoverLoadType.Gripper THEN 
				 fbPuncherSeparateStation.P_List_Switch_Input_N.AddMover(GVL.g_Movers[index].std);
			  END_IF
			  
			 
		END_FOR

	
			nExecutingSequence := nExecutingSequence+1;

15: 		// set process mode 
		 	 FOR index := 1 TO GVL.gc_NumberStations DO
 			GVL.g_Stations[index].P_eProcessMode := E_ProcessMode.Production;		   
	 	   END_FOR
			
				nExecutingSequence := nExecutingSequence+1;

16:			//process method
			Communication.g_Com_GlobalState.OUT.InCycle:=TRUE; 
			fbPuncherStation.Process();
			fbPuncherSeparateStation.Process();
			
			nExecutingSequence := 0;

20,30: 

		 	 FOR index := 1 TO GVL.gc_NumberStations DO
 			GVL.g_Stations[index].P_eProcessMode := E_ProcessMode.None;		   
	 	   END_FOR
	

		FOR index := 1 TO gvl. g_nMoverCount DO
		
		GVL.g_Movers[index].ManualMovement(FALSE);
		END_FOR

	nExecutingSequence := 0;

// test movement

	
